FUNCTION_BLOCK "Qm"   // FB10, SCL
{ S7_Optimized_Access := 'FALSE' }
VERSION : 0.1
// Массовый расход
   VAR_INPUT
      Enable : Bool;   // Наличие параметра
      "a" : Real;   // Коэффициент расхода
      Ksh : Real;   // Поправочный коэффициент на шероховатость трубопровода
      Kp : Real;   // Поправочный коэффициент на неостроту входной кромки диафрагмы
      d : Real;   // Диаметр сужающего устройства при рабочих условиях (мм)
      ro : Real;   // Плотность среды в рабочих условиях (кг/м3)
      dP : Real;   // Перепад давления в рабочих условиях (кПа)
   END_VAR
   VAR_OUTPUT
      Value : Real;   // Значение массового расхода (т/ч)
   END_VAR
BEGIN
   (*Расход массового расхода (т/ч)*)
   IF #Enable THEN
       #Value := (#"a" * #Ksh * #Kp * 3.1415926 * SQR(#d / 1000) / 4) * SQRT(2 * #dP * 1000* #ro) * 3.6;
   ELSE
       #Value := 0;
   END_IF;
   IF #dP < 0 THEN
       #Value := 0;
   END_IF;
END_FUNCTION_BLOCK

FUNCTION_BLOCK "Qm_steam"   // FB11, SCL
{ S7_Optimized_Access := 'FALSE' }
VERSION : 0.1
// Массовый расход пара
   VAR_INPUT
      Enable : Bool;   // Наличие параметра
      "a" : Real;   // Коэффициент расхода
      Ksh : Real;   // Поправочный коэффициент на шероховатость трубопровода
      Kp : Real;   // Поправочный коэффициент на неостроту входной кромки диафрагмы
      d : Real;   // Диаметр сужающего устройства при рабочих условиях (мм)
      Dtrub : Real;   // Диаметр трубопровода при рабочих условиях (мм)
      k : Real;   // Показатель адиабаты
      ro : Real;   // Плотность среды в рабочих условиях (кг/м3)
      dP : Real;   // Перепад давления в рабочих условиях (кПа)
      P : Real;   // Давление в рабочих условиях (кПа)
   END_VAR
   VAR_OUTPUT
      Value : Real;   // Значение массового расхода (т/ч)
   END_VAR
   VAR
      "E" : Real;   // Коэффициент расширения
      B4 : Real;   // Относительный диаметр сужающего устройства (в 4 степени)
   END_VAR
BEGIN
   IF #Enable THEN
       (*Расчет относительного диаметра сужающего устройства (в 4 степени)*)
       #B4 := (#d /#Dtrub) ** 4;
       (*Расчет коэффициента расширения*)
       #"E" := 1 - ((0.351 + (0.256 * #B4) + (0.93 * SQR(#B4))) * (1 - ((1 - (#dP / #P)) ** (1 / #k))));
       #Value:= 0.25 * SQR(#d / 1000) * 3.1415926 * #"a" * #Ksh * #Kp * #"E" * SQRT(2 * #dP * #ro) * 3.6;
   ELSE
       #Value := 0;
   END_IF;
   IF #dP <= 0 OR #P <= 0 THEN
       #Value := 0;
   END_IF;
END_FUNCTION_BLOCK

FUNCTION_BLOCK "ro"   // FB12, SCL
{ S7_Optimized_Access := 'FALSE' }
VERSION : 0.1
// Расчет плотности
   VAR_INPUT
      P : Array[1..10] of Real;   // Давление (МПа)
      T : Array[1..20] of Real;   // Температура (град С)
      PT : Array[1..10, 1..20] of Real;   // Удельный объем (л/кг)
      Px : Real;   // Текущее давление (МПа)
      Tx : Real;   // Текущая температура (град С)
   END_VAR
   VAR_OUTPUT
      ro : Real;   // Значение удельной плотности (кг/м3)
   END_VAR
   VAR
      Pmin : Int;   // Нижняя граница текущего диапазона давления
      Pmax : Int;   // Верхняя граница текущего диапазона давления
      Tmin : Int;   // Нижняя граница текущего диапазона температуры
      Tmax : Int;   // Верхняя граница текущего диапазона температуры
      Pmin_Tmin : Real;   // Значение Pmin_Tmin рабочей области
      Pmin_Tmax : Real;   // Значение Pmin_Tmax рабочей области
      Pmax_Tmin : Real;   // Значение Pmax_Tmin рабочей области
      Pmax_Tmax : Real;   // Значение Pmax_Tmax рабочей области
      Px_Tmin : Real;   // Значение Px_Tmin суженной рабочей области
      Px_Tmax : Real;   // Значение Px_Tmax суженной рабочей области
      K_Px_Tmin : Real;
      B_Px_Tmin : Real;
      K_Px_Tmax : Real;
      B_Px_Tmax : Real;
      Px_Tx : Real;   // Искомое значение удельного объема (л/кг)
      K_Px_Tx : Real;
      B_Px_Tx : Real;
   END_VAR
BEGIN
   (*определение текущего диапазона давления*)
   IF #Px <= #P[2] THEN
       #Pmin := 1;
       #Pmax := 2;
   END_IF;
   IF #P[2] < #Px AND #Px <= #P[3] THEN
       #Pmin := 2;
       #Pmax := 3;
   END_IF;
   IF #P[3] < #Px AND #Px <= #P[4] THEN
       #Pmin := 3;
       #Pmax := 4;
   END_IF;
   IF #P[4] < #Px AND #Px <= #P[5] THEN
       #Pmin := 4;
       #Pmax := 5;
   END_IF;
   IF #P[5] < #Px AND #Px <= #P[6] THEN
       #Pmin := 5;
       #Pmax := 6;
   END_IF;
   IF #P[6] < #Px AND #Px <= #P[7] THEN
       #Pmin := 6;
       #Pmax := 7;
   END_IF;
   IF #P[7] < #Px AND #Px <= #P[8] THEN
       #Pmin := 7;
       #Pmax := 8;
   END_IF;
   IF #P[8] < #Px AND #Px <= #P[9] THEN
       #Pmin := 8;
       #Pmax := 9;
   END_IF;
   IF #P[9] < #Px THEN
       #Pmin := 9;
       #Pmax := 10;
   END_IF;

   (*определение текущего диапазона температуры*)
   IF #Tx <= #T[2] THEN
       #Tmin := 1;
       #Tmax := 2;
   END_IF;
   IF #T[2] < #Tx AND #Tx <= #T[3] THEN
       #Tmin := 2;
       #Tmax := 3;
   END_IF;
   IF #T[3] < #Tx AND #Tx <= #T[4] THEN
       #Tmin := 3;
       #Tmax := 4;
   END_IF;
   IF #T[4] < #Tx AND #Tx <= #T[5] THEN
       #Tmin := 4;
       #Tmax := 5;
   END_IF;
   IF #T[5] < #Tx AND #Tx <= #T[6] THEN
       #Tmin := 5;
       #Tmax := 6;
   END_IF;
   IF #T[6] < #Tx AND #Tx <= #T[7] THEN
       #Tmin := 6;
       #Tmax := 7;
   END_IF;
   IF #T[7] < #Tx AND #Tx <= #T[8] THEN
       #Tmin := 7;
       #Tmax := 8;
   END_IF;
   IF #T[8] < #Tx AND #Tx <= #T[9] THEN
       #Tmin := 8;
       #Tmax := 9;
   END_IF;
   IF #T[9] < #Tx AND #Tx <= #T[10] THEN
       #Tmin := 9;
       #Tmax := 10;
   END_IF;
   IF #T[10] < #Tx AND #Tx <= #T[11] THEN
       #Tmin := 10;
       #Tmax := 11;
   END_IF;
   IF #T[11] < #Tx AND #Tx <= #T[12] THEN
       #Tmin := 11;
       #Tmax := 12;
   END_IF;
   IF #T[12] < #Tx AND #Tx <= #T[13] THEN
       #Tmin := 12;
       #Tmax := 13;
   END_IF;
   IF #T[13] < #Tx AND #Tx <= #T[14] THEN
       #Tmin := 13;
       #Tmax := 14;
   END_IF;
   IF #T[14] < #Tx AND #Tx <= #T[15] THEN
       #Tmin := 14;
       #Tmax := 15;
   END_IF;
   IF #T[15] < #Tx AND #Tx <= #T[16] THEN
       #Tmin := 15;
       #Tmax := 16;
   END_IF;
   IF #T[16] < #Tx AND #Tx <= #T[17] THEN
       #Tmin := 16;
       #Tmax := 17;
   END_IF;
   IF #T[17] < #Tx AND #Tx <= #T[18] THEN
       #Tmin := 17;
       #Tmax := 18;
   END_IF;
   IF #T[18] < #Tx AND #Tx <= #T[19] THEN
       #Tmin := 18;
       #Tmax := 19;
   END_IF;
   IF #T[19] < #Tx THEN
       #Tmin := 19;
       #Tmax := 20;
   END_IF;

   (*определение рабочей области*)
   #Pmin_Tmin := #PT[#Pmin, #Tmin];
   #Pmin_Tmax := #PT[#Pmin, #Tmax];
   #Pmax_Tmin := #PT[#Pmax, #Tmin];
   #Pmax_Tmax := #PT[#Pmax, #Tmax];

   (*определение суженной по давлению рабочей области*)
   #K_Px_Tmin := (#Pmax_Tmin - #Pmin_Tmin) / (#P[#Pmax] - #P[#Pmin]);
   #B_Px_Tmin := #Pmin_Tmin - #K_Px_Tmin * #P[#Pmin];
   #Px_Tmin := #K_Px_Tmin * #Px + #B_Px_Tmin;

   #K_Px_Tmax := (#Pmax_Tmax - #Pmin_Tmax) / (#P[#Pmax] - #P[#Pmin]);
   #B_Px_Tmax := #Pmin_Tmax - #K_Px_Tmax * #P[#Pmin];
   #Px_Tmax := #K_Px_Tmax * #Px + #B_Px_Tmax;

   (*определение искомого значения удельного объема*)
   #K_Px_Tx := (#Px_Tmax - #Px_Tmin) / (#T[#Tmax] - #T[#Tmin]);
   #B_Px_Tx := #Px_Tmin - #K_Px_Tx * #T[#Tmin];
   #Px_Tx := #K_Px_Tx * #Tx + #B_Px_Tx;

   (*определение значения удельной плотности*)
   #ro := 1000 / #Px_Tx;
END_FUNCTION_BLOCK

FUNCTION_BLOCK "Qs"   // FB13, SCL
{ S7_Optimized_Access := 'FALSE' }
VERSION : 0.1
// Расход приведенный к стандартным условиям (нм3/ч)
   VAR_INPUT
      P : Real;   // Давление в рабочих условиях (Па)
      Q : Real;   // Объемный расход измеренный (м3/ч)
      T : Real;   // Температура в рабочих условиях (град С)
      ro_c : Real;   // Плотность при стандартных условиях (кг/м3)
      Xa : Real;   // молярная/объемная доля азота (в долях от 1)
      Xy : Real;   // молярная/объемная доля диоксида углерода (в долях от 1)
   END_VAR
   VAR_OUTPUT
      Qs : Real;   // Объемный расход приведенный к стандартным условиям (нм3/ч)
   END_VAR
   VAR
      K : Real;   // коэффициент сжимаемости
      Z : Real;   // фактор сжимаемости при рабочих условиях
      Zc : Real;   // фактор сжимаемости при стандартных условиях
      Tpk : Real;
      Ppk : Real;
      Ta : Real;
      Pa : Real;
      dTa : Real;
      F : Real;   // Корректирующий множитель
      Theta1 : Real;
      Theta0 : Real;
      B0 : Real;
      B1 : Real;
      B2 : Real;
   END_VAR
BEGIN
   (*расчет фактора сжимаемости при стандартных условиях*)
   #Zc := 1 - SQR(0.0741*#ro_c-0.006-0.063*#Xa-0.0575*#Xy);

   (*расчет фактора сжимаемости при рабочих условиях*)
   #Tpk:=88.25*(0.9915+1.759*#ro_c-#Xy-1.681*#Xa);
   #Ppk := 2.9585 * (1.608-0.05994*#ro_c+#Xy-0.392*#Xa);

   #Ta := 0.71892 * ((#T + 273.15)/ #Tpk) + 0.0007;
   #Pa := 0.6714 * (#P / (1000000*#Ppk)) + 0.0147;

   #dTa := #Ta - 1.09;

   //расчет корректирующего множителя
   IF 0 <= #Pa AND #Pa <= 2 AND 0 <= #dTa AND #dTa <= 0.3 THEN
       #F := (0.00075 * (#Pa ** 2.3)) / (2.718281828459045 ** (20 * #dTa)) + 0.0011*SQRT(#dTa)*SQR((#Pa*(2.17-#Pa+1.4*SQRT(#dTa))));
   END_IF;
   IF 0 <= #Pa AND #Pa < 1.3 AND -0.25 <= #dTa AND #dTa < 0 THEN
       #F := 0.00075 * (#Pa ** 2.3) * (2 - (2.718281828459045 ** (20 * #dTa))) + 1.317 * #Pa * (1.69 - SQR(#Pa)) * (#dTa ** 4);
   END_IF;
   IF 1.3 <= #Pa AND #Pa < 2 AND -0.21 <= #dTa AND #dTa < 0 THEN
       #F := 0.00075 * (#Pa ** 2.3) * (2 - (2.718281828459045 ** (20 * #dTa)))+0.455*#Pa*(1.3-#Pa)*(4.0195200-SQR(#Pa))*(#dTa*(0.03249+18.028*SQR(#dTa))+SQR(#dTa)*(2.0167+SQR(#dTa)*(42.844+200*SQR(#dTa))));
   END_IF;

   #Theta1 := (#Ta ** 5) / (SQR(#Ta)*(6.60756*#Ta-4.42646)+3.22706);
   #Theta0 := ((SQR(#Ta)*(1.77218-0.8879*#Ta)+0.305131) * #Theta1) / (#Ta ** 4);
   #B1 := ((2 * #Theta1) / 3) - SQR(#Theta0);
   #B0 := #Theta0 * (#Theta1 - SQR(#Theta0)) + 0.1 * #Theta1 * #Pa * (#F - 1);
   #B2 := (#B0 + SQRT(SQR(#B0) + #B1 ** 3)) ** (0.333334);

   #Z := ((1+(0.00132/(#Ta**3.25))) / ((#B1/#B2)-#B2+#Theta0)) * (#Pa / 10);

   (*расчет коэффициента сжимаемости*)
   #K := #Z / #Zc;

   (*расчет объемного расхода приведенного к стандартным условиям (нм3/ч)*)
   #Qs := ((#P+101325) * 293.15 * #Q) / (101325 * (#T + 273.15) * #K);
END_FUNCTION_BLOCK

FUNCTION "Read_inputs" : Void   // FC1, SCL
{ S7_Optimized_Access := 'TRUE' }
VERSION : 0.1
BEGIN
   (*ЧТЕНИЕ ВХОДОВ*)
   (*Чтение аналоговых входов*)
   //Температура питательной воды перед экономайзером
   "T_water_before_economizer"();
   //Температура питательной воды после экономайзера
   "T_water_after_economizer"();
   //Перепад давления питательной воды на котел
   "dP_water_boiler"();
   //Давление питательной воды до регулятора
   "P_water_before_regul"();
   //Давление питательной воды после регулятора
   "P_water_after_regul"();
   //Перепад давления пара в магистраль
   "dP_steam"();
   //Давление пара в барабане
   "P_steam"();
   //Разрежение в топке котла
   "dP_furnace_boiler"();
   //Давление газа между ПЗК-1 и ПЗК-2
   "P_gas_between_PZK1_and_PZK2"();
   //Давление газа перед горелкой
   "P_gas_before_burner"();
   //Давление воздуха к горелке
   "P_air_burner"();
   //Положение рег. заслонки питательной воды на котел
   "ZRW_position"();
   //Положение рег. заслонки газа перед котлом
   "ZRG_position"();
   //Положение направл. аппарата вентилятора
   "NAV_position"();
   //Положение направл. аппарата дымососа
   "NAD_position"();
   //Температура уходящих дымовых газов  перед экономайзером
   "T_exhaust_gas_before_economizer"();
   //Температура уходящих дымовых газов  после экономайзера
   "T_exhaust_gas_after_economizer"();
   //Разрежение в дымоходе перед экономайзером
   "dP_exhaust_gas_before_economizer"();
   //Разрежение в дымоходе после экономайзера
   "dP_exhaust_gas_after_economizer"();
   //Давление газа перед БГ
   "P_gas_before_BG"();
   //Температура газа перед БГ
   "T_gas_before_BG"();
   //Давление пара в магистраль
   "P_steam_pipe"();
   //Температура пара в магистраль
   "T_steam"();
   //Текущее значение частоты ПЧ вентилятора
   "DV_current_frequency"();
   //Текущее значение частоты ПЧ дымососа
   "DS_current_frequency"();
   //Перепад давления на измерительной колонке 
   "dP_water_level"();
   //Уровень воды в измерительной колонке
   "L_water_level"(LL_ADC_new := "dP_water_level".LL_ADC_new,
                   HL_ADC_new := "dP_water_level".HL_ADC_new,
                   Apply_new_limit := "dP_water_level".Apply_new_limit);
   //Уровень воды в барабане
   "L_water"(LL_sensor_new := "L_water_level".LL_sensor_new + "Technology".Offset_level_water,
             HL_sensor_new := "L_water_level".HL_sensor_new + "Technology".Offset_level_water,
             LL_ADC_new := "dP_water_level".LL_ADC_new,
             HL_ADC_new := "dP_water_level".HL_ADC_new,
             Apply_new_limit := "dP_water_level".Apply_new_limit);

   (*Чтение дискретных входов*)
   //Наличие пламени горелки
   "Burner_flame"();
   //Наличие пламени запальника горелки
   "Igniter_flame"();
   //Клапан безопасности закрыт
   "KB_close"();
   //Клапан опрессовки открыт
   "KO_open"();
   //Клапан запальника открыт
   "KZ_open"();
   //ПЗК-1 горелки открыт
   "PZK1_open"();
   //ПЗК-2 горелки не закрыт
   "PZK2_not_close"();
   //Давление газа перед БГ мин.
   "P_gas_before_BG_min"();
   //Давление газа перед БГ макс.
   "P_gas_before_BG_max"();
   //Давление воздуха перед горелкой мин.
   "P_air_before_burner_min"();
   //Давление газа перед горелкой мин.
   "P_gas_before_burner_min"();
   //Давление газа перед горелкой макс.
   "P_gas_before_burner_max"();
   //Регулирующая заслонка газа открыта
   "ZRG_open"();
   //Регулирующая заслонка газа закрыта
   "ZRG_close"();
   //Регулирующая заслонка газа среднее
   "ZRG_middle"();
   //Регулирующая заслонка газа. БРУ в положении "Авт"
   "ZRG_avto"();
   //НАВ открыт
   "NAV_open"();
   //НАВ закрыт
   "NAV_close"();
   //НАВ среднее
   "NAV_middle"();
   //НАВ. БРУ в положении "Авт"
   "NAV_avto"();
   //НАД открыт
   "NAD_open"();
   //НАД закрыт
   "NAD_close"();
   //НАД среднее
   "NAD_middle"();
   //НАД. БРУ в положении "Авт"
   "NAD_avto"();
   //ПЗК-2 горелки открыт
   "PZK2_open"();
   //Разрежение в топке котла мин.
   "dP_furnace_boiler_min"();
   //Давление питательной воды после регулятора мин.
   "P_water_after_regul_min"();
   //Давление пара в барабане макс.
   "P_steam_max"();
   //Уровень воды в барабане мин.
   "L_water_min"();
   //Уровень воды в барабане макс.
   "L_water_max"();
   //Вызов к шкафу электропитания
   "Call_power_supply_cabinet"();
   //Авария ПЧ ДВ
   "DV_Invertor_alarm"();
   //Режим работы ДВ «Местный»
   "DV_local_control"();
   //Режим работы ДВ «Дистанционный»
   "DV_dist_control"();
   //Режим "СЕТЬ" ДВ
   "DV_powergrid_mode"();
   //Режим "ПЧ" ДВ
   "DV_invertor_mode"();
   //Автомат работы ДВ от ПЧ включен
   "DV_invertor_QF_on"();
   //Автомат работы ДВ от сети включен
   "DV_powergrid_QF_on"();
   //Включен ДВ от ПЧ
   "DV_invertor_on"();
   //Включен ДВ от сети
   "DV_powergrid_on"();
   //Нет напряжения сети ШУД ДВ
   "DV_no_voltage"();
   //Авария ПЧ ДС
   "DS_Invertor_alarm"();
   //Режим работы ДС «Местный»
   "DS_local_control"();
   //Режим работы ДC «Дистанционный»
   "DS_dist_control"();
   //Режим "СЕТЬ" ДC
   "DS_powergrid_mode"();
   //Режим "ПЧ" ДС
   "DS_invertor_mode"();
   //Автомат работы ДС от ПЧ включен
   "DS_invertor_QF_on"();
   //Автомат работы ДС от сети включен
   "DS_powergrid_QF_on"();
   //Включен ДС от ПЧ
   "DS_invertor_on"();
   //Включен ДС от сети
   "DS_powergrid_on"();
   //Нет напряжения сети ШУД ДС
   "DS_no_voltage"();
   //Загазованность СО I порог
   "CO_1"();
   //Загазованность СО II порог
   "CO_2"();
   //Загазованность CH4 порог
   "CH4"();
   //Кнопка СТОП
   "Btn_STOP"();
   //Кнопка Вентиляция
   "Btn_Ventilation"();
   //Кнопка Розжиг
   "Btn_Ignition"();
   //Кнопка Сброс звука / Проверка звука
   "Btn_Sound"();
   //Регулирующая заслонка питательной воды на котел открыта
   "ZRW_open"();
   //Регулирующая заслонка питательной воды на котел закрыта
   "ZRW_close"();
   //Регулирующая заслонка питательной воды на котел среднее
   "ZRW_middle"();
   //Регулирующая заслонка питательной воды на котел. БРУ в положении "Авт"
   "ZRW_avto"();
   //Питание контроллера от ИБП
   "Power_PLC_from_UPS"();
   //Заряд батареи ИБП низкий
   "UPS_Low_charge"();
   //ЗРГ Напряжение в норме
   "ZRG_voltage_ok"();
   //НАВ Напряжение в норме
   "NAV_voltage_ok"();
   //НАД Напряжение в норме
   "NAD_voltage_ok"();
   //ЗРВ Напряжение в норме
   "ZRW_voltage_ok"();
   //Контроль питания сети ~400В 1ШЭУ
   "SHEU_voltage_ok"();
   //ЗДГ перед БГ. не открыта
   "ZDG_no_open"();
   //ЗДГ перед БГ. не закрыта
   "ZDG_no_close"();
   //ЗДГ перед БГ. ход открытие
   "ZDG_opening"();
   //ЗДГ перед БГ. ход закрытие
   "ZDG_closing"();
   //ЗДГ перед БГ. Напряжение в норме
   "ZDG_voltage_ok"();
   //ЗДСВ перед котлом. не открыта
   "ZDSV_before_boiler_no_open"();
   //ЗДСВ перед котлом. не закрыта
   "ZDSV_before_boiler_no_close"();
   //ЗДСВ перед котлом. ход открытие
   "ZDSV_before_boiler_opening"();
   //ЗДСВ перед котлом. ход закрытие
   "ZDSV_before_boiler_closing"();
   //ЗДСВ перед котлом. Напряжение в норме
   "ZDSV_before_boiler_voltage_ok"();
   //ЗДСВ перед котлом. ограничитель крутящего момента
   "ZDSV_before_boiler_limit_rotational_moment"();
   //ГПЗ. не открыта
   "GPZ_no_open"();
   //ГПЗ. не закрыта
   "GPZ_no_close"();
   //ГПЗ. ход открытие
   "GPZ_opening"();
   //ГПЗ. ход закрытие
   "GPZ_closing"();
   //ГПЗ. Напряжение в норме
   "GPZ_voltage_ok"();
   //ГПЗ. ограничитель крутящего момента
   "GPZ_limit_rotational_moment"();

   (*Контроль питания ~400В резервной горелки, статус «Работа на дизтопливе»

   Режим работы резервной горелки

   Блокировка пламени резервной горелки

   Режим “Большое пламя» резервной горелки*)

   //Расход газа (м3/ч)
   //"Q_gas".scale_unit := (293.15 * INT_TO_REAL("Technology".Q_gas_scale_unit) * ("P_gas_before_BG".Value/1000.0 + "Technology".P_atm))/(0.101325*(273.15 + "T_gas_before_BG".Value)*"Technology".K_gas);
   "Q_gas"();

   //Расход газа приведенного к стандартным условиям (нм3/ч)
   "Qs_gas"(P := "P_gas_before_BG".Value * 1000,
            Q := "Q_gas".moment_consumption,
            T := "T_gas_before_BG".Value);

   //Массовый расход воды
   "Q_water"(dP := "dP_water_boiler".Value);

   //плотность пара
   "ro_steam"(Px := ("P_steam_pipe".Value) / 10,
              Tx := "T_steam".Value);

   //Массовый расход пара
   IF "GPZ_no_close".Value THEN
       "Q_steam"(dP := "dP_steam".Value * 1000,
                 P := ("P_steam_pipe".Value + 1) * 100000,
                 ro := "ro_steam".ro);
   ELSE
       "Q_steam"(dP := 0 * 1000,
                 P := ("P_steam_pipe".Value + 1) * 100000,
                 ro := "ro_steam".ro);
   END_IF;
   "Q1_water".Value := ("Qs_gas".Qs * "Q1_water".Calorie * "Q1_water".KPD) / ("Q1_water"."E" * 1000);

   (*настройка датчиков уровня*)
   "dP_main" := ((("dP_water_boiler".HL_sensor - "dP_water_boiler".LL_sensor) / INT_TO_REAL(27648 - 0)) * INT_TO_REAL("Module03Chanel5_AI")) + "dP_water_boiler".LL_sensor;
   "L_main" := ((("L_water".HL_sensor - "L_water".LL_sensor) / INT_TO_REAL(0 - 27648)) * INT_TO_REAL("Module03Chanel5_AI")) + "L_water".HL_sensor;
   "Current_main" := (((20 - 4) / (INT_TO_REAL(27648 - 0))) * (INT_TO_REAL("Module03Chanel5_AI"))) + 4;

   "dP_res" := ((("dP_water_boiler".HL_sensor - "dP_water_boiler".LL_sensor) / INT_TO_REAL(27648 - 0)) * INT_TO_REAL("Module04Chanel5_AI")) + "dP_water_boiler".LL_sensor;
   "L_res" := ((("L_water".HL_sensor - "L_water".LL_sensor) / INT_TO_REAL(0 - 27648)) * INT_TO_REAL("Module04Chanel5_AI")) + "L_water".HL_sensor;
   "Current_res" := (((20 - 4) / (INT_TO_REAL(27648 - 0))) * (INT_TO_REAL("Module04Chanel5_AI"))) + 4;

   //подмена дискретных входов
   "Module12Chanel1_DI" := "Module12Chanel1_DO";
   "Module12Chanel2_DI" := "Module12Chanel2_DO";
   "Module12Chanel3_DI" := "Module12Chanel3_DO";
   "Module12Chanel4_DI" := "Module12Chanel4_DO";
   "Module12Chanel5_DI" := "Module12Chanel5_DO";
   "Module12Chanel6_DI" := "Module12Chanel6_DO";
   "Module12Chanel7_DI" := "Module12Chanel7_DO";
   "Module12Chanel8_DI" := "Module12Chanel8_DO";
   "Module12Chanel9_DI" := "Module12Chanel9_DO";
   "Module12Chanel10_DI" := "Module12Chanel10_DO";
   "Module12Chanel11_DI" := "Module12Chanel11_DO";
   "Module12Chanel12_DI" := "Module12Chanel12_DO";
   "Module12Chanel13_DI" := "Module12Chanel13_DO";
   "Module12Chanel14_DI" := "Module12Chanel14_DO";
   "Module12Chanel15_DI" := "Module12Chanel15_DO";
   "Module12Chanel16_DI" := "Module12Chanel16_DO";
END_FUNCTION

FUNCTION "read_discret" : Bool   // FC2, SCL
{ S7_Optimized_Access := 'TRUE' }
AUTHOR : Dmitriy_Petrov
VERSION : 0.1
// Функция чтения дискретного параметра
   VAR_INPUT
      Invert : Bool;   // Инвертирование сигнала
   END_VAR
   VAR_IN_OUT
      N_module : USInt;   // № модуля (начиная с 1)
      N_chanel : USInt;   // № канала (начиная с 1)
   END_VAR
   VAR_TEMP
      Signal : Bool;   // Значение сигнала
   END_VAR
   // Ret_Val : Текущее значение
BEGIN
   (*проверка правильности введеного значения № Модуля*)
   IF #N_module < 1 OR #N_module > 25 THEN
       #N_module := 0;
   END_IF;

   (*проверка правильности введеного значения № Канала*)
   IF #N_module = 0 THEN
       #N_chanel := 0;
   ELSE
       IF #N_chanel < 1 OR #N_chanel > 16 THEN
           #N_chanel := 0;
       END_IF;
   END_IF;

   (*считывание и обработка дискретного сигнала с выбранного канала*)
   CASE #N_module OF
       1:  // Модуль 1
           CASE #N_chanel OF
               1:
                   #Signal := "Module01Chanel1_DI";   //Канал 1
               2:
                   #Signal := "Module01Chanel2_DI";   //Канал 2
               3:
                   #Signal := "Module01Chanel3_DI";   //Канал 3
               4:
                   #Signal := "Module01Chanel4_DI";   //Канал 4
               5:
                   #Signal := "Module01Chanel5_DI";   //Канал 5
               6:
                   #Signal := "Module01Chanel6_DI";   //Канал 6
               7:
                   #Signal := "Module01Chanel7_DI";   //Канал 7
               8:
                   #Signal := "Module01Chanel8_DI";   //Канал 8
               9:
                   #Signal := "Module01Chanel9_DI";   //Канал 9
               10:
                   #Signal := "Module01Chanel10_DI";  //Канал 10
               11:
                   #Signal := "Module01Chanel11_DI";  //Канал 11
               12:
                   #Signal := "Module01Chanel12_DI";  //Канал 12
               13:
                   #Signal := "Module01Chanel13_DI";  //Канал 13
               14:
                   #Signal := "Module01Chanel14_DI";  //Канал 14
               15:
                   #Signal := "Module01Chanel15_DI";  //Канал 15
               16:
                   #Signal := "Module01Chanel16_DI";  //Канал 16
               ELSE
                   #Signal := FALSE;
           END_CASE;
       2:  // Модуль 2
           CASE #N_chanel OF
               1:
                   #Signal := "Module02Chanel1_DI";   //Канал 1
               2:
                   #Signal := "Module02Chanel2_DI";   //Канал 2
               3:
                   #Signal := "Module02Chanel3_DI";   //Канал 3
               4:
                   #Signal := "Module02Chanel4_DI";   //Канал 4
               5:
                   #Signal := "Module02Chanel5_DI";   //Канал 5
               6:
                   #Signal := "Module02Chanel6_DI";   //Канал 6
               7:
                   #Signal := "Module02Chanel7_DI";   //Канал 7
               8:
                   #Signal := "Module02Chanel8_DI";   //Канал 8
               9:
                   #Signal := "Module02Chanel9_DI";   //Канал 9
               10:
                   #Signal := "Module02Chanel10_DI";  //Канал 10
               11:
                   #Signal := "Module02Chanel11_DI";  //Канал 11
               12:
                   #Signal := "Module02Chanel12_DI";  //Канал 12
               13:
                   #Signal := "Module02Chanel13_DI";  //Канал 13
               14:
                   #Signal := "Module02Chanel14_DI";  //Канал 14
               15:
                   #Signal := "Module02Chanel15_DI";  //Канал 15
               16:
                   #Signal := "Module02Chanel16_DI";  //Канал 16
               ELSE
                   #Signal := FALSE;
           END_CASE;
       3:  // Модуль 3
           CASE #N_chanel OF
               1:
                   #Signal := "Module03Chanel1_DI";   //Канал 1
               2:
                   #Signal := "Module03Chanel2_DI";   //Канал 2
               3:
                   #Signal := "Module03Chanel3_DI";   //Канал 3
               4:
                   #Signal := "Module03Chanel4_DI";   //Канал 4
               5:
                   #Signal := "Module03Chanel5_DI";   //Канал 5
               6:
                   #Signal := "Module03Chanel6_DI";   //Канал 6
               7:
                   #Signal := "Module03Chanel7_DI";   //Канал 7
               8:
                   #Signal := "Module03Chanel8_DI";   //Канал 8
               9:
                   #Signal := "Module03Chanel9_DI";   //Канал 9
               10:
                   #Signal := "Module03Chanel10_DI";  //Канал 10
               11:
                   #Signal := "Module03Chanel11_DI";  //Канал 11
               12:
                   #Signal := "Module03Chanel12_DI";  //Канал 12
               13:
                   #Signal := "Module03Chanel13_DI";  //Канал 13
               14:
                   #Signal := "Module03Chanel14_DI";  //Канал 14
               15:
                   #Signal := "Module03Chanel15_DI";  //Канал 15
               16:
                   #Signal := "Module03Chanel16_DI";  //Канал 16
               ELSE
                   #Signal := FALSE;
           END_CASE;
       4:  // Модуль 4
           CASE #N_chanel OF
               1:
                   #Signal := "Module04Chanel1_DI";   //Канал 1
               2:
                   #Signal := "Module04Chanel2_DI";   //Канал 2
               3:
                   #Signal := "Module04Chanel3_DI";   //Канал 3
               4:
                   #Signal := "Module04Chanel4_DI";   //Канал 4
               5:
                   #Signal := "Module04Chanel5_DI";   //Канал 5
               6:
                   #Signal := "Module04Chanel6_DI";   //Канал 6
               7:
                   #Signal := "Module04Chanel7_DI";   //Канал 7
               8:
                   #Signal := "Module04Chanel8_DI";   //Канал 8
               9:
                   #Signal := "Module04Chanel9_DI";   //Канал 9
               10:
                   #Signal := "Module04Chanel10_DI";  //Канал 10
               11:
                   #Signal := "Module04Chanel11_DI";  //Канал 11
               12:
                   #Signal := "Module04Chanel12_DI";  //Канал 12
               13:
                   #Signal := "Module04Chanel13_DI";  //Канал 13
               14:
                   #Signal := "Module04Chanel14_DI";  //Канал 14
               15:
                   #Signal := "Module04Chanel15_DI";  //Канал 15
               16:
                   #Signal := "Module04Chanel16_DI";  //Канал 16
               ELSE
                   #Signal := FALSE;
           END_CASE;
       5:  // Модуль 5
           CASE #N_chanel OF
               1:
                   #Signal := "Module05Chanel1_DI";   //Канал 1
               2:
                   #Signal := "Module05Chanel2_DI";   //Канал 2
               3:
                   #Signal := "Module05Chanel3_DI";   //Канал 3
               4:
                   #Signal := "Module05Chanel4_DI";   //Канал 4
               5:
                   #Signal := "Module05Chanel5_DI";   //Канал 5
               6:
                   #Signal := "Module05Chanel6_DI";   //Канал 6
               7:
                   #Signal := "Module05Chanel7_DI";   //Канал 7
               8:
                   #Signal := "Module05Chanel8_DI";   //Канал 8
               9:
                   #Signal := "Module05Chanel9_DI";   //Канал 9
               10:
                   #Signal := "Module05Chanel10_DI";  //Канал 10
               11:
                   #Signal := "Module05Chanel11_DI";  //Канал 11
               12:
                   #Signal := "Module05Chanel12_DI";  //Канал 12
               13:
                   #Signal := "Module05Chanel13_DI";  //Канал 13
               14:
                   #Signal := "Module05Chanel14_DI";  //Канал 14
               15:
                   #Signal := "Module05Chanel15_DI";  //Канал 15
               16:
                   #Signal := "Module05Chanel16_DI";  //Канал 16
               ELSE
                   #Signal := FALSE;
           END_CASE;
       6:  // Модуль 6
           CASE #N_chanel OF
               1:
                   #Signal := "Module06Chanel1_DI";   //Канал 1
               2:
                   #Signal := "Module06Chanel2_DI";   //Канал 2
               3:
                   #Signal := "Module06Chanel3_DI";   //Канал 3
               4:
                   #Signal := "Module06Chanel4_DI";   //Канал 4
               5:
                   #Signal := "Module06Chanel5_DI";   //Канал 5
               6:
                   #Signal := "Module06Chanel6_DI";   //Канал 6
               7:
                   #Signal := "Module06Chanel7_DI";   //Канал 7
               8:
                   #Signal := "Module06Chanel8_DI";   //Канал 8
               9:
                   #Signal := "Module06Chanel9_DI";   //Канал 9
               10:
                   #Signal := "Module06Chanel10_DI";  //Канал 10
               11:
                   #Signal := "Module06Chanel11_DI";  //Канал 11
               12:
                   #Signal := "Module06Chanel12_DI";  //Канал 12
               13:
                   #Signal := "Module06Chanel13_DI";  //Канал 13
               14:
                   #Signal := "Module06Chanel14_DI";  //Канал 14
               15:
                   #Signal := "Module06Chanel15_DI";  //Канал 15
               16:
                   #Signal := "Module06Chanel16_DI";  //Канал 16
               ELSE
                   #Signal := FALSE;
           END_CASE;
       7:  // Модуль 7
           CASE #N_chanel OF
               1:
                   #Signal := "Module07Chanel1_DI";   //Канал 1
               2:
                   #Signal := "Module07Chanel2_DI";   //Канал 2
               3:
                   #Signal := "Module07Chanel3_DI";   //Канал 3
               4:
                   #Signal := "Module07Chanel4_DI";   //Канал 4
               5:
                   #Signal := "Module07Chanel5_DI";   //Канал 5
               6:
                   #Signal := "Module07Chanel6_DI";   //Канал 6
               7:
                   #Signal := "Module07Chanel7_DI";   //Канал 7
               8:
                   #Signal := "Module07Chanel8_DI";   //Канал 8
               9:
                   #Signal := "Module07Chanel9_DI";   //Канал 9
               10:
                   #Signal := "Module07Chanel10_DI";  //Канал 10
               11:
                   #Signal := "Module07Chanel11_DI";  //Канал 11
               12:
                   #Signal := "Module07Chanel12_DI";  //Канал 12
               13:
                   #Signal := "Module07Chanel13_DI";  //Канал 13
               14:
                   #Signal := "Module07Chanel14_DI";  //Канал 14
               15:
                   #Signal := "Module07Chanel15_DI";  //Канал 15
               16:
                   #Signal := "Module07Chanel16_DI";  //Канал 16
               ELSE
                   #Signal := FALSE;
           END_CASE;
       8:  // Модуль 8
           CASE #N_chanel OF
               1:
                   #Signal := "Module08Chanel1_DI";   //Канал 1
               2:
                   #Signal := "Module08Chanel2_DI";   //Канал 2
               3:
                   #Signal := "Module08Chanel3_DI";   //Канал 3
               4:
                   #Signal := "Module08Chanel4_DI";   //Канал 4
               5:
                   #Signal := "Module08Chanel5_DI";   //Канал 5
               6:
                   #Signal := "Module08Chanel6_DI";   //Канал 6
               7:
                   #Signal := "Module08Chanel7_DI";   //Канал 7
               8:
                   #Signal := "Module08Chanel8_DI";   //Канал 8
               9:
                   #Signal := "Module08Chanel9_DI";   //Канал 9
               10:
                   #Signal := "Module08Chanel10_DI";  //Канал 10
               11:
                   #Signal := "Module08Chanel11_DI";  //Канал 11
               12:
                   #Signal := "Module08Chanel12_DI";  //Канал 12
               13:
                   #Signal := "Module08Chanel13_DI";  //Канал 13
               14:
                   #Signal := "Module08Chanel14_DI";  //Канал 14
               15:
                   #Signal := "Module08Chanel15_DI";  //Канал 15
               16:
                   #Signal := "Module08Chanel16_DI";  //Канал 16
               ELSE
                   #Signal := FALSE;
           END_CASE;
       9:  // Модуль 9
           CASE #N_chanel OF
               1:
                   #Signal := "Module09Chanel1_DI";   //Канал 1
               2:
                   #Signal := "Module09Chanel2_DI";   //Канал 2
               3:
                   #Signal := "Module09Chanel3_DI";   //Канал 3
               4:
                   #Signal := "Module09Chanel4_DI";   //Канал 4
               5:
                   #Signal := "Module09Chanel5_DI";   //Канал 5
               6:
                   #Signal := "Module09Chanel6_DI";   //Канал 6
               7:
                   #Signal := "Module09Chanel7_DI";   //Канал 7
               8:
                   #Signal := "Module09Chanel8_DI";   //Канал 8
               9:
                   #Signal := "Module09Chanel9_DI";   //Канал 9
               10:
                   #Signal := "Module09Chanel10_DI";  //Канал 10
               11:
                   #Signal := "Module09Chanel11_DI";  //Канал 11
               12:
                   #Signal := "Module09Chanel12_DI";  //Канал 12
               13:
                   #Signal := "Module09Chanel13_DI";  //Канал 13
               14:
                   #Signal := "Module09Chanel14_DI";  //Канал 14
               15:
                   #Signal := "Module09Chanel15_DI";  //Канал 15
               16:
                   #Signal := "Module09Chanel16_DI";  //Канал 16
               ELSE
                   #Signal := FALSE;
           END_CASE;
       10:  // Модуль 10
           CASE #N_chanel OF
               1:
                   #Signal := "Module10Chanel1_DI";   //Канал 1
               2:
                   #Signal := "Module10Chanel2_DI";   //Канал 2
               3:
                   #Signal := "Module10Chanel3_DI";   //Канал 3
               4:
                   #Signal := "Module10Chanel4_DI";   //Канал 4
               5:
                   #Signal := "Module10Chanel5_DI";   //Канал 5
               6:
                   #Signal := "Module10Chanel6_DI";   //Канал 6
               7:
                   #Signal := "Module10Chanel7_DI";   //Канал 7
               8:
                   #Signal := "Module10Chanel8_DI";   //Канал 8
               9:
                   #Signal := "Module10Chanel9_DI";   //Канал 9
               10:
                   #Signal := "Module10Chanel10_DI";  //Канал 10
               11:
                   #Signal := "Module10Chanel11_DI";  //Канал 11
               12:
                   #Signal := "Module10Chanel12_DI";  //Канал 12
               13:
                   #Signal := "Module10Chanel13_DI";  //Канал 13
               14:
                   #Signal := "Module10Chanel14_DI";  //Канал 14
               15:
                   #Signal := "Module10Chanel15_DI";  //Канал 15
               16:
                   #Signal := "Module10Chanel16_DI";  //Канал 16
               ELSE
                   #Signal := FALSE;
           END_CASE;
       11:  // Модуль 11
           CASE #N_chanel OF
               1:
                   #Signal := "Module11Chanel1_DI";   //Канал 1
               2:
                   #Signal := "Module11Chanel2_DI";   //Канал 2
               3:
                   #Signal := "Module11Chanel3_DI";   //Канал 3
               4:
                   #Signal := "Module11Chanel4_DI";   //Канал 4
               5:
                   #Signal := "Module11Chanel5_DI";   //Канал 5
               6:
                   #Signal := "Module11Chanel6_DI";   //Канал 6
               7:
                   #Signal := "Module11Chanel7_DI";   //Канал 7
               8:
                   #Signal := "Module11Chanel8_DI";   //Канал 8
               9:
                   #Signal := "Module11Chanel9_DI";   //Канал 9
               10:
                   #Signal := "Module11Chanel10_DI";  //Канал 10
               11:
                   #Signal := "Module11Chanel11_DI";  //Канал 11
               12:
                   #Signal := "Module11Chanel12_DI";  //Канал 12
               13:
                   #Signal := "Module11Chanel13_DI";  //Канал 13
               14:
                   #Signal := "Module11Chanel14_DI";  //Канал 14
               15:
                   #Signal := "Module11Chanel15_DI";  //Канал 15
               16:
                   #Signal := "Module11Chanel16_DI";  //Канал 16
               ELSE
                   #Signal := FALSE;
           END_CASE;
       12:  // Модуль 12
           CASE #N_chanel OF
               1:
                   #Signal := "Module12Chanel1_DI";   //Канал 1
               2:
                   #Signal := "Module12Chanel2_DI";   //Канал 2
               3:
                   #Signal := "Module12Chanel3_DI";   //Канал 3
               4:
                   #Signal := "Module12Chanel4_DI";   //Канал 4
               5:
                   #Signal := "Module12Chanel5_DI";   //Канал 5
               6:
                   #Signal := "Module12Chanel6_DI";   //Канал 6
               7:
                   #Signal := "Module12Chanel7_DI";   //Канал 7
               8:
                   #Signal := "Module12Chanel8_DI";   //Канал 8
               9:
                   #Signal := "Module12Chanel9_DI";   //Канал 9
               10:
                   #Signal := "Module12Chanel10_DI";  //Канал 10
               11:
                   #Signal := "Module12Chanel11_DI";  //Канал 11
               12:
                   #Signal := "Module12Chanel12_DI";  //Канал 12
               13:
                   #Signal := "Module12Chanel13_DI";  //Канал 13
               14:
                   #Signal := "Module12Chanel14_DI";  //Канал 14
               15:
                   #Signal := "Module12Chanel15_DI";  //Канал 15
               16:
                   #Signal := "Module12Chanel16_DI";  //Канал 16
               ELSE
                   #Signal := FALSE;
           END_CASE;
       13:  // Модуль 13
           CASE #N_chanel OF
               1:
                   #Signal := "Module13Chanel1_DI";   //Канал 1
               2:
                   #Signal := "Module13Chanel2_DI";   //Канал 2
               3:
                   #Signal := "Module13Chanel3_DI";   //Канал 3
               4:
                   #Signal := "Module13Chanel4_DI";   //Канал 4
               5:
                   #Signal := "Module13Chanel5_DI";   //Канал 5
               6:
                   #Signal := "Module13Chanel6_DI";   //Канал 6
               7:
                   #Signal := "Module13Chanel7_DI";   //Канал 7
               8:
                   #Signal := "Module13Chanel8_DI";   //Канал 8
               9:
                   #Signal := "Module13Chanel9_DI";   //Канал 9
               10:
                   #Signal := "Module13Chanel10_DI";  //Канал 10
               11:
                   #Signal := "Module13Chanel11_DI";  //Канал 11
               12:
                   #Signal := "Module13Chanel12_DI";  //Канал 12
               13:
                   #Signal := "Module13Chanel13_DI";  //Канал 13
               14:
                   #Signal := "Module13Chanel14_DI";  //Канал 14
               15:
                   #Signal := "Module13Chanel15_DI";  //Канал 15
               16:
                   #Signal := "Module13Chanel16_DI";  //Канал 16
               ELSE
                   #Signal := FALSE;
           END_CASE;
       14:  // Модуль 14
           CASE #N_chanel OF
               1:
                   #Signal := "Module14Chanel1_DI";   //Канал 1
               2:
                   #Signal := "Module14Chanel2_DI";   //Канал 2
               3:
                   #Signal := "Module14Chanel3_DI";   //Канал 3
               4:
                   #Signal := "Module14Chanel4_DI";   //Канал 4
               5:
                   #Signal := "Module14Chanel5_DI";   //Канал 5
               6:
                   #Signal := "Module14Chanel6_DI";   //Канал 6
               7:
                   #Signal := "Module14Chanel7_DI";   //Канал 7
               8:
                   #Signal := "Module14Chanel8_DI";   //Канал 8
               9:
                   #Signal := "Module14Chanel9_DI";   //Канал 9
               10:
                   #Signal := "Module14Chanel10_DI";  //Канал 10
               11:
                   #Signal := "Module14Chanel11_DI";  //Канал 11
               12:
                   #Signal := "Module14Chanel12_DI";  //Канал 12
               13:
                   #Signal := "Module14Chanel13_DI";  //Канал 13
               14:
                   #Signal := "Module14Chanel14_DI";  //Канал 14
               15:
                   #Signal := "Module14Chanel15_DI";  //Канал 15
               16:
                   #Signal := "Module14Chanel16_DI";  //Канал 16
               ELSE
                   #Signal := FALSE;
           END_CASE;
       15:  // Модуль 15
           CASE #N_chanel OF
               1:
                   #Signal := "Module15Chanel1_DI";   //Канал 1
               2:
                   #Signal := "Module15Chanel2_DI";   //Канал 2
               3:
                   #Signal := "Module15Chanel3_DI";   //Канал 3
               4:
                   #Signal := "Module15Chanel4_DI";   //Канал 4
               5:
                   #Signal := "Module15Chanel5_DI";   //Канал 5
               6:
                   #Signal := "Module15Chanel6_DI";   //Канал 6
               7:
                   #Signal := "Module15Chanel7_DI";   //Канал 7
               8:
                   #Signal := "Module15Chanel8_DI";   //Канал 8
               9:
                   #Signal := "Module15Chanel9_DI";   //Канал 9
               10:
                   #Signal := "Module15Chanel10_DI";  //Канал 10
               11:
                   #Signal := "Module15Chanel11_DI";  //Канал 11
               12:
                   #Signal := "Module15Chanel12_DI";  //Канал 12
               13:
                   #Signal := "Module15Chanel13_DI";  //Канал 13
               14:
                   #Signal := "Module15Chanel14_DI";  //Канал 14
               15:
                   #Signal := "Module15Chanel15_DI";  //Канал 15
               16:
                   #Signal := "Module15Chanel16_DI";  //Канал 16
               ELSE
                   #Signal := FALSE;
           END_CASE;
       16:  // Модуль 16
           CASE #N_chanel OF
               1:
                   #Signal := "Module16Chanel1_DI";   //Канал 1
               2:
                   #Signal := "Module16Chanel2_DI";   //Канал 2
               3:
                   #Signal := "Module16Chanel3_DI";   //Канал 3
               4:
                   #Signal := "Module16Chanel4_DI";   //Канал 4
               5:
                   #Signal := "Module16Chanel5_DI";   //Канал 5
               6:
                   #Signal := "Module16Chanel6_DI";   //Канал 6
               7:
                   #Signal := "Module16Chanel7_DI";   //Канал 7
               8:
                   #Signal := "Module16Chanel8_DI";   //Канал 8
               9:
                   #Signal := "Module16Chanel9_DI";   //Канал 9
               10:
                   #Signal := "Module16Chanel10_DI";  //Канал 10
               11:
                   #Signal := "Module16Chanel11_DI";  //Канал 11
               12:
                   #Signal := "Module16Chanel12_DI";  //Канал 12
               13:
                   #Signal := "Module16Chanel13_DI";  //Канал 13
               14:
                   #Signal := "Module16Chanel14_DI";  //Канал 14
               15:
                   #Signal := "Module16Chanel15_DI";  //Канал 15
               16:
                   #Signal := "Module16Chanel16_DI";  //Канал 16
               ELSE
                   #Signal := FALSE;
           END_CASE;
       17:  // Модуль 17
           CASE #N_chanel OF
               1:
                   #Signal := "Module17Chanel1_DI";   //Канал 1
               2:
                   #Signal := "Module17Chanel2_DI";   //Канал 2
               3:
                   #Signal := "Module17Chanel3_DI";   //Канал 3
               4:
                   #Signal := "Module17Chanel4_DI";   //Канал 4
               5:
                   #Signal := "Module17Chanel5_DI";   //Канал 5
               6:
                   #Signal := "Module17Chanel6_DI";   //Канал 6
               7:
                   #Signal := "Module17Chanel7_DI";   //Канал 7
               8:
                   #Signal := "Module17Chanel8_DI";   //Канал 8
               9:
                   #Signal := "Module17Chanel9_DI";   //Канал 9
               10:
                   #Signal := "Module17Chanel10_DI";  //Канал 10
               11:
                   #Signal := "Module17Chanel11_DI";  //Канал 11
               12:
                   #Signal := "Module17Chanel12_DI";  //Канал 12
               13:
                   #Signal := "Module17Chanel13_DI";  //Канал 13
               14:
                   #Signal := "Module17Chanel14_DI";  //Канал 14
               15:
                   #Signal := "Module17Chanel15_DI";  //Канал 15
               16:
                   #Signal := "Module17Chanel16_DI";  //Канал 16
               ELSE
                   #Signal := FALSE;
           END_CASE;
       18:  // Модуль 18
           CASE #N_chanel OF
               1:
                   #Signal := "Module18Chanel1_DI";   //Канал 1
               2:
                   #Signal := "Module18Chanel2_DI";   //Канал 2
               3:
                   #Signal := "Module18Chanel3_DI";   //Канал 3
               4:
                   #Signal := "Module18Chanel4_DI";   //Канал 4
               5:
                   #Signal := "Module18Chanel5_DI";   //Канал 5
               6:
                   #Signal := "Module18Chanel6_DI";   //Канал 6
               7:
                   #Signal := "Module18Chanel7_DI";   //Канал 7
               8:
                   #Signal := "Module18Chanel8_DI";   //Канал 8
               9:
                   #Signal := "Module18Chanel9_DI";   //Канал 9
               10:
                   #Signal := "Module18Chanel10_DI";  //Канал 10
               11:
                   #Signal := "Module18Chanel11_DI";  //Канал 11
               12:
                   #Signal := "Module18Chanel12_DI";  //Канал 12
               13:
                   #Signal := "Module18Chanel13_DI";  //Канал 13
               14:
                   #Signal := "Module18Chanel14_DI";  //Канал 14
               15:
                   #Signal := "Module18Chanel15_DI";  //Канал 15
               16:
                   #Signal := "Module18Chanel16_DI";  //Канал 16
               ELSE
                   #Signal := FALSE;
           END_CASE;
       19:  // Модуль 19
           CASE #N_chanel OF
               1:
                   #Signal := "Module19Chanel1_DI";   //Канал 1
               2:
                   #Signal := "Module19Chanel2_DI";   //Канал 2
               3:
                   #Signal := "Module19Chanel3_DI";   //Канал 3
               4:
                   #Signal := "Module19Chanel4_DI";   //Канал 4
               5:
                   #Signal := "Module19Chanel5_DI";   //Канал 5
               6:
                   #Signal := "Module19Chanel6_DI";   //Канал 6
               7:
                   #Signal := "Module19Chanel7_DI";   //Канал 7
               8:
                   #Signal := "Module19Chanel8_DI";   //Канал 8
               9:
                   #Signal := "Module19Chanel9_DI";   //Канал 9
               10:
                   #Signal := "Module19Chanel10_DI";  //Канал 10
               11:
                   #Signal := "Module19Chanel11_DI";  //Канал 11
               12:
                   #Signal := "Module19Chanel12_DI";  //Канал 12
               13:
                   #Signal := "Module19Chanel13_DI";  //Канал 13
               14:
                   #Signal := "Module19Chanel14_DI";  //Канал 14
               15:
                   #Signal := "Module19Chanel15_DI";  //Канал 15
               16:
                   #Signal := "Module19Chanel16_DI";  //Канал 16
               ELSE
                   #Signal := FALSE;
           END_CASE;
       20:  // Модуль 20
           CASE #N_chanel OF
               1:
                   #Signal := "Module20Chanel1_DI";   //Канал 1
               2:
                   #Signal := "Module20Chanel2_DI";   //Канал 2
               3:
                   #Signal := "Module20Chanel3_DI";   //Канал 3
               4:
                   #Signal := "Module20Chanel4_DI";   //Канал 4
               5:
                   #Signal := "Module20Chanel5_DI";   //Канал 5
               6:
                   #Signal := "Module20Chanel6_DI";   //Канал 6
               7:
                   #Signal := "Module20Chanel7_DI";   //Канал 7
               8:
                   #Signal := "Module20Chanel8_DI";   //Канал 8
               9:
                   #Signal := "Module20Chanel9_DI";   //Канал 9
               10:
                   #Signal := "Module20Chanel10_DI";  //Канал 10
               11:
                   #Signal := "Module20Chanel11_DI";  //Канал 11
               12:
                   #Signal := "Module20Chanel12_DI";  //Канал 12
               13:
                   #Signal := "Module20Chanel13_DI";  //Канал 13
               14:
                   #Signal := "Module20Chanel14_DI";  //Канал 14
               15:
                   #Signal := "Module20Chanel15_DI";  //Канал 15
               16:
                   #Signal := "Module20Chanel16_DI";  //Канал 16
               ELSE
                   #Signal := FALSE;
           END_CASE;
       21:  // Модуль 21
           CASE #N_chanel OF
               1:
                   #Signal := "Module21Chanel1_DI";   //Канал 1
               2:
                   #Signal := "Module21Chanel2_DI";   //Канал 2
               3:
                   #Signal := "Module21Chanel3_DI";   //Канал 3
               4:
                   #Signal := "Module21Chanel4_DI";   //Канал 4
               5:
                   #Signal := "Module21Chanel5_DI";   //Канал 5
               6:
                   #Signal := "Module21Chanel6_DI";   //Канал 6
               7:
                   #Signal := "Module21Chanel7_DI";   //Канал 7
               8:
                   #Signal := "Module21Chanel8_DI";   //Канал 8
               9:
                   #Signal := "Module21Chanel9_DI";   //Канал 9
               10:
                   #Signal := "Module21Chanel10_DI";  //Канал 10
               11:
                   #Signal := "Module21Chanel11_DI";  //Канал 11
               12:
                   #Signal := "Module21Chanel12_DI";  //Канал 12
               13:
                   #Signal := "Module21Chanel13_DI";  //Канал 13
               14:
                   #Signal := "Module21Chanel14_DI";  //Канал 14
               15:
                   #Signal := "Module21Chanel15_DI";  //Канал 15
               16:
                   #Signal := "Module21Chanel16_DI";  //Канал 16
               ELSE
                   #Signal := FALSE;
           END_CASE;
       22:  // Модуль 22
           CASE #N_chanel OF
               1:
                   #Signal := "Module22Chanel1_DI";   //Канал 1
               2:
                   #Signal := "Module22Chanel2_DI";   //Канал 2
               3:
                   #Signal := "Module22Chanel3_DI";   //Канал 3
               4:
                   #Signal := "Module22Chanel4_DI";   //Канал 4
               5:
                   #Signal := "Module22Chanel5_DI";   //Канал 5
               6:
                   #Signal := "Module22Chanel6_DI";   //Канал 6
               7:
                   #Signal := "Module22Chanel7_DI";   //Канал 7
               8:
                   #Signal := "Module22Chanel8_DI";   //Канал 8
               9:
                   #Signal := "Module22Chanel9_DI";   //Канал 9
               10:
                   #Signal := "Module22Chanel10_DI";  //Канал 10
               11:
                   #Signal := "Module22Chanel11_DI";  //Канал 11
               12:
                   #Signal := "Module22Chanel12_DI";  //Канал 12
               13:
                   #Signal := "Module22Chanel13_DI";  //Канал 13
               14:
                   #Signal := "Module22Chanel14_DI";  //Канал 14
               15:
                   #Signal := "Module22Chanel15_DI";  //Канал 15
               16:
                   #Signal := "Module22Chanel16_DI";  //Канал 16
               ELSE
                   #Signal := FALSE;
           END_CASE;
       23:  // Модуль 23
           CASE #N_chanel OF
               1:
                   #Signal := "Module23Chanel1_DI";   //Канал 1
               2:
                   #Signal := "Module23Chanel2_DI";   //Канал 2
               3:
                   #Signal := "Module23Chanel3_DI";   //Канал 3
               4:
                   #Signal := "Module23Chanel4_DI";   //Канал 4
               5:
                   #Signal := "Module23Chanel5_DI";   //Канал 5
               6:
                   #Signal := "Module23Chanel6_DI";   //Канал 6
               7:
                   #Signal := "Module23Chanel7_DI";   //Канал 7
               8:
                   #Signal := "Module23Chanel8_DI";   //Канал 8
               9:
                   #Signal := "Module23Chanel9_DI";   //Канал 9
               10:
                   #Signal := "Module23Chanel10_DI";  //Канал 10
               11:
                   #Signal := "Module23Chanel11_DI";  //Канал 11
               12:
                   #Signal := "Module23Chanel12_DI";  //Канал 12
               13:
                   #Signal := "Module23Chanel13_DI";  //Канал 13
               14:
                   #Signal := "Module23Chanel14_DI";  //Канал 14
               15:
                   #Signal := "Module23Chanel15_DI";  //Канал 15
               16:
                   #Signal := "Module23Chanel16_DI";  //Канал 16
               ELSE
                   #Signal := FALSE;
           END_CASE;
       24:  // Модуль 24
           CASE #N_chanel OF
               1:
                   #Signal := "Module24Chanel1_DI";   //Канал 1
               2:
                   #Signal := "Module24Chanel2_DI";   //Канал 2
               3:
                   #Signal := "Module24Chanel3_DI";   //Канал 3
               4:
                   #Signal := "Module24Chanel4_DI";   //Канал 4
               5:
                   #Signal := "Module24Chanel5_DI";   //Канал 5
               6:
                   #Signal := "Module24Chanel6_DI";   //Канал 6
               7:
                   #Signal := "Module24Chanel7_DI";   //Канал 7
               8:
                   #Signal := "Module24Chanel8_DI";   //Канал 8
               9:
                   #Signal := "Module24Chanel9_DI";   //Канал 9
               10:
                   #Signal := "Module24Chanel10_DI";  //Канал 10
               11:
                   #Signal := "Module24Chanel11_DI";  //Канал 11
               12:
                   #Signal := "Module24Chanel12_DI";  //Канал 12
               13:
                   #Signal := "Module24Chanel13_DI";  //Канал 13
               14:
                   #Signal := "Module24Chanel14_DI";  //Канал 14
               15:
                   #Signal := "Module24Chanel15_DI";  //Канал 15
               16:
                   #Signal := "Module24Chanel16_DI";  //Канал 16
               ELSE
                   #Signal := FALSE;
           END_CASE;
       25:  // Модуль 25
           CASE #N_chanel OF
               1:
                   #Signal := "Module25Chanel1_DI";   //Канал 1
               2:
                   #Signal := "Module25Chanel2_DI";   //Канал 2
               3:
                   #Signal := "Module25Chanel3_DI";   //Канал 3
               4:
                   #Signal := "Module25Chanel4_DI";   //Канал 4
               5:
                   #Signal := "Module25Chanel5_DI";   //Канал 5
               6:
                   #Signal := "Module25Chanel6_DI";   //Канал 6
               7:
                   #Signal := "Module25Chanel7_DI";   //Канал 7
               8:
                   #Signal := "Module25Chanel8_DI";   //Канал 8
               9:
                   #Signal := "Module25Chanel9_DI";   //Канал 9
               10:
                   #Signal := "Module25Chanel10_DI";  //Канал 10
               11:
                   #Signal := "Module25Chanel11_DI";  //Канал 11
               12:
                   #Signal := "Module25Chanel12_DI";  //Канал 12
               13:
                   #Signal := "Module25Chanel13_DI";  //Канал 13
               14:
                   #Signal := "Module25Chanel14_DI";  //Канал 14
               15:
                   #Signal := "Module25Chanel15_DI";  //Канал 15
               16:
                   #Signal := "Module25Chanel16_DI";  //Канал 16
               ELSE
                   #Signal := FALSE;
           END_CASE;
       ELSE
           #Signal := FALSE;
   END_CASE;
   IF NOT #Invert THEN
       #read_discret:= #Signal;
   ELSE
       #read_discret:= NOT #Signal;
   END_IF;
END_FUNCTION

FUNCTION "read_4_20" : Real   // FC3, SCL
{ S7_Optimized_Access := 'TRUE' }
AUTHOR : Dmitriy_Petrov
VERSION : 0.1
// Функция чтения сигнала 4-20mA
   VAR_INPUT
      LL_sensor : Real;   // Нижний предел датчика в физической величине
      HL_sensor : Real;   // Верхний предел датчика в физической величине
      LL_ADC : Int;   // Нижний предел АЦП
      HL_ADC : Int;   // Верхний предел АЦП
   END_VAR
   VAR_OUTPUT
      Current : Real;   // Значение тока
      error_sensor : Bool;   // Неисправность датчика
   END_VAR
   VAR_IN_OUT
      N_module : USInt;   // № модуля (начиная с 1)
      N_chanel : USInt;   // № канала (начиная с 1)
      ADC : Int;   // Текущий код АЦП
   END_VAR
   VAR_TEMP
      K : Real;   // Коэффициент К
      "B" : Real;   // Коэффициент B
   END_VAR
BEGIN
   (*проверка правильности введенного значения № Модуля*)
   IF #N_module < 1 OR #N_module > 25 THEN
       #N_module := 0;
   END_IF;

   (*проверка правильности введенного значения № Канала*)
   IF #N_module = 0 THEN
       #N_chanel := 0;
   ELSE
       IF #N_chanel < 1 OR #N_chanel > 8 THEN
           #N_chanel := 0;
       END_IF;
   END_IF;

   (*считывание кода АЦП выбранного канала*)
   CASE #N_module OF
       1:  // Модуль 1
           CASE #N_chanel OF
               1:
                   #ADC := "Module01Chanel1_AI";   //Канал 1
               2:
                   #ADC := "Module01Chanel2_AI";   //Канал 2
               3:
                   #ADC := "Module01Chanel3_AI";   //Канал 3
               4:
                   #ADC := "Module01Chanel4_AI";   //Канал 4
               5:
                   #ADC := "Module01Chanel5_AI";   //Канал 5
               6:
                   #ADC := "Module01Chanel6_AI";   //Канал 6
               7:
                   #ADC := "Module01Chanel7_AI";   //Канал 7
               8:
                   #ADC := "Module01Chanel8_AI";   //Канал 8
               ELSE
                   #ADC := 0;
           END_CASE;
       2:  // Модуль 2
           CASE #N_chanel OF
               1:
                   #ADC := "Module02Chanel1_AI";   //Канал 1
               2:
                   #ADC := "Module02Chanel2_AI";   //Канал 2
               3:
                   #ADC := "Module02Chanel3_AI";   //Канал 3
               4:
                   #ADC := "Module02Chanel4_AI";   //Канал 4
               5:
                   #ADC := "Module02Chanel5_AI";   //Канал 5
               6:
                   #ADC := "Module02Chanel6_AI";   //Канал 6
               7:
                   #ADC := "Module02Chanel7_AI";   //Канал 7
               8:
                   #ADC := "Module02Chanel8_AI";   //Канал 8
               ELSE
                   #ADC := 0;
           END_CASE;
       3:  // Модуль 3
           CASE #N_chanel OF
               1:
                   #ADC := "Module03Chanel1_AI";   //Канал 1
               2:
                   #ADC := "Module03Chanel2_AI";   //Канал 2
               3:
                   #ADC := "Module03Chanel3_AI";   //Канал 3
               4:
                   #ADC := "Module03Chanel4_AI";   //Канал 4
               5:
                   #ADC := "Module03Chanel5_AI";   //Канал 5
               6:
                   #ADC := "Module03Chanel6_AI";   //Канал 6
               7:
                   #ADC := "Module03Chanel7_AI";   //Канал 7
               8:
                   #ADC := "Module03Chanel8_AI";   //Канал 8
               ELSE
                   #ADC := 0;
           END_CASE;
       4:  // Модуль 4
           CASE #N_chanel OF
               1:
                   #ADC := "Module04Chanel1_AI";   //Канал 1
               2:
                   #ADC := "Module04Chanel2_AI";   //Канал 2
               3:
                   #ADC := "Module04Chanel3_AI";   //Канал 3
               4:
                   #ADC := "Module04Chanel4_AI";   //Канал 4
               5:
                   #ADC := "Module04Chanel5_AI";   //Канал 5
               6:
                   #ADC := "Module04Chanel6_AI";   //Канал 6
               7:
                   #ADC := "Module04Chanel7_AI";   //Канал 7
               8:
                   #ADC := "Module04Chanel8_AI";   //Канал 8
               ELSE
                   #ADC := 0;
           END_CASE;
       5:  // Модуль 5
           CASE #N_chanel OF
               1:
                   #ADC := "Module05Chanel1_AI";   //Канал 1
               2:
                   #ADC := "Module05Chanel2_AI";   //Канал 2
               3:
                   #ADC := "Module05Chanel3_AI";   //Канал 3
               4:
                   #ADC := "Module05Chanel4_AI";   //Канал 4
               5:
                   #ADC := "Module05Chanel5_AI";   //Канал 5
               6:
                   #ADC := "Module05Chanel6_AI";   //Канал 6
               7:
                   #ADC := "Module05Chanel7_AI";   //Канал 7
               8:
                   #ADC := "Module05Chanel8_AI";   //Канал 8
               ELSE
                   #ADC := 0;
           END_CASE;
       6:  // Модуль 6
           CASE #N_chanel OF
               1:
                   #ADC := "Module06Chanel1_AI";   //Канал 1
               2:
                   #ADC := "Module06Chanel2_AI";   //Канал 2
               3:
                   #ADC := "Module06Chanel3_AI";   //Канал 3
               4:
                   #ADC := "Module06Chanel4_AI";   //Канал 4
               5:
                   #ADC := "Module06Chanel5_AI";   //Канал 5
               6:
                   #ADC := "Module06Chanel6_AI";   //Канал 6
               7:
                   #ADC := "Module06Chanel7_AI";   //Канал 7
               8:
                   #ADC := "Module06Chanel8_AI";   //Канал 8
               ELSE
                   #ADC := 0;
           END_CASE;
       7:  // Модуль 7
           CASE #N_chanel OF
               1:
                   #ADC := "Module07Chanel1_AI";   //Канал 1
               2:
                   #ADC := "Module07Chanel2_AI";   //Канал 2
               3:
                   #ADC := "Module07Chanel3_AI";   //Канал 3
               4:
                   #ADC := "Module07Chanel4_AI";   //Канал 4
               5:
                   #ADC := "Module07Chanel5_AI";   //Канал 5
               6:
                   #ADC := "Module07Chanel6_AI";   //Канал 6
               7:
                   #ADC := "Module07Chanel7_AI";   //Канал 7
               8:
                   #ADC := "Module07Chanel8_AI";   //Канал 8
               ELSE
                   #ADC := 0;
           END_CASE;
       8:  // Модуль 8
           CASE #N_chanel OF
               1:
                   #ADC := "Module08Chanel1_AI";   //Канал 1
               2:
                   #ADC := "Module08Chanel2_AI";   //Канал 2
               3:
                   #ADC := "Module08Chanel3_AI";   //Канал 3
               4:
                   #ADC := "Module08Chanel4_AI";   //Канал 4
               5:
                   #ADC := "Module08Chanel5_AI";   //Канал 5
               6:
                   #ADC := "Module08Chanel6_AI";   //Канал 6
               7:
                   #ADC := "Module08Chanel7_AI";   //Канал 7
               8:
                   #ADC := "Module08Chanel8_AI";   //Канал 8
               ELSE
                   #ADC := 0;
           END_CASE;
       9:  // Модуль 9
           CASE #N_chanel OF
               1:
                   #ADC := "Module09Chanel1_AI";   //Канал 1
               2:
                   #ADC := "Module09Chanel2_AI";   //Канал 2
               3:
                   #ADC := "Module09Chanel3_AI";   //Канал 3
               4:
                   #ADC := "Module09Chanel4_AI";   //Канал 4
               5:
                   #ADC := "Module09Chanel5_AI";   //Канал 5
               6:
                   #ADC := "Module09Chanel6_AI";   //Канал 6
               7:
                   #ADC := "Module09Chanel7_AI";   //Канал 7
               8:
                   #ADC := "Module09Chanel8_AI";   //Канал 8
               ELSE
                   #ADC := 0;
           END_CASE;
       10:  // Модуль 10
           CASE #N_chanel OF
               1:
                   #ADC := "Module10Chanel1_AI";   //Канал 1
               2:
                   #ADC := "Module10Chanel2_AI";   //Канал 2
               3:
                   #ADC := "Module10Chanel3_AI";   //Канал 3
               4:
                   #ADC := "Module10Chanel4_AI";   //Канал 4
               5:
                   #ADC := "Module10Chanel5_AI";   //Канал 5
               6:
                   #ADC := "Module10Chanel6_AI";   //Канал 6
               7:
                   #ADC := "Module10Chanel7_AI";   //Канал 7
               8:
                   #ADC := "Module10Chanel8_AI";   //Канал 8
               ELSE
                   #ADC := 0;
           END_CASE;
       11:  // Модуль 11
           CASE #N_chanel OF
               1:
                   #ADC := "Module11Chanel1_AI";   //Канал 1
               2:
                   #ADC := "Module11Chanel2_AI";   //Канал 2
               3:
                   #ADC := "Module11Chanel3_AI";   //Канал 3
               4:
                   #ADC := "Module11Chanel4_AI";   //Канал 4
               5:
                   #ADC := "Module11Chanel5_AI";   //Канал 5
               6:
                   #ADC := "Module11Chanel6_AI";   //Канал 6
               7:
                   #ADC := "Module11Chanel7_AI";   //Канал 7
               8:
                   #ADC := "Module11Chanel8_AI";   //Канал 8
               ELSE
                   #ADC := 0;
           END_CASE;
       12:  // Модуль 12
           CASE #N_chanel OF
               1:
                   #ADC := "Module12Chanel1_AI";   //Канал 1
               2:
                   #ADC := "Module12Chanel2_AI";   //Канал 2
               3:
                   #ADC := "Module12Chanel3_AI";   //Канал 3
               4:
                   #ADC := "Module12Chanel4_AI";   //Канал 4
               5:
                   #ADC := "Module12Chanel5_AI";   //Канал 5
               6:
                   #ADC := "Module12Chanel6_AI";   //Канал 6
               7:
                   #ADC := "Module12Chanel7_AI";   //Канал 7
               8:
                   #ADC := "Module12Chanel8_AI";   //Канал 8
               ELSE
                   #ADC := 0;
           END_CASE;
       13:  // Модуль 13
           CASE #N_chanel OF
               1:
                   #ADC := "Module13Chanel1_AI";   //Канал 1
               2:
                   #ADC := "Module13Chanel2_AI";   //Канал 2
               3:
                   #ADC := "Module13Chanel3_AI";   //Канал 3
               4:
                   #ADC := "Module13Chanel4_AI";   //Канал 4
               5:
                   #ADC := "Module13Chanel5_AI";   //Канал 5
               6:
                   #ADC := "Module13Chanel6_AI";   //Канал 6
               7:
                   #ADC := "Module13Chanel7_AI";   //Канал 7
               8:
                   #ADC := "Module13Chanel8_AI";   //Канал 8
               ELSE
                   #ADC := 0;
           END_CASE;
       14:  // Модуль 14
           CASE #N_chanel OF
               1:
                   #ADC := "Module14Chanel1_AI";   //Канал 1
               2:
                   #ADC := "Module14Chanel2_AI";   //Канал 2
               3:
                   #ADC := "Module14Chanel3_AI";   //Канал 3
               4:
                   #ADC := "Module14Chanel4_AI";   //Канал 4
               5:
                   #ADC := "Module14Chanel5_AI";   //Канал 5
               6:
                   #ADC := "Module14Chanel6_AI";   //Канал 6
               7:
                   #ADC := "Module14Chanel7_AI";   //Канал 7
               8:
                   #ADC := "Module14Chanel8_AI";   //Канал 8
               ELSE
                   #ADC := 0;
           END_CASE;
       15:  // Модуль 15
           CASE #N_chanel OF
               1:
                   #ADC := "Module15Chanel1_AI";   //Канал 1
               2:
                   #ADC := "Module15Chanel2_AI";   //Канал 2
               3:
                   #ADC := "Module15Chanel3_AI";   //Канал 3
               4:
                   #ADC := "Module15Chanel4_AI";   //Канал 4
               5:
                   #ADC := "Module15Chanel5_AI";   //Канал 5
               6:
                   #ADC := "Module15Chanel6_AI";   //Канал 6
               7:
                   #ADC := "Module15Chanel7_AI";   //Канал 7
               8:
                   #ADC := "Module15Chanel8_AI";   //Канал 8
               ELSE
                   #ADC := 0;
           END_CASE;
       16:  // Модуль 16
           CASE #N_chanel OF
               1:
                   #ADC := "Module16Chanel1_AI";   //Канал 1
               2:
                   #ADC := "Module16Chanel2_AI";   //Канал 2
               3:
                   #ADC := "Module16Chanel3_AI";   //Канал 3
               4:
                   #ADC := "Module16Chanel4_AI";   //Канал 4
               5:
                   #ADC := "Module16Chanel5_AI";   //Канал 5
               6:
                   #ADC := "Module16Chanel6_AI";   //Канал 6
               7:
                   #ADC := "Module16Chanel7_AI";   //Канал 7
               8:
                   #ADC := "Module16Chanel8_AI";   //Канал 8
               ELSE
                   #ADC := 0;
           END_CASE;
       17:  // Модуль 17
           CASE #N_chanel OF
               1:
                   #ADC := "Module17Chanel1_AI";   //Канал 1
               2:
                   #ADC := "Module17Chanel2_AI";   //Канал 2
               3:
                   #ADC := "Module17Chanel3_AI";   //Канал 3
               4:
                   #ADC := "Module17Chanel4_AI";   //Канал 4
               5:
                   #ADC := "Module17Chanel5_AI";   //Канал 5
               6:
                   #ADC := "Module17Chanel6_AI";   //Канал 6
               7:
                   #ADC := "Module17Chanel7_AI";   //Канал 7
               8:
                   #ADC := "Module17Chanel8_AI";   //Канал 8
               ELSE
                   #ADC := 0;
           END_CASE;
       18:  // Модуль 18
           CASE #N_chanel OF
               1:
                   #ADC := "Module18Chanel1_AI";   //Канал 1
               2:
                   #ADC := "Module18Chanel2_AI";   //Канал 2
               3:
                   #ADC := "Module18Chanel3_AI";   //Канал 3
               4:
                   #ADC := "Module18Chanel4_AI";   //Канал 4
               5:
                   #ADC := "Module18Chanel5_AI";   //Канал 5
               6:
                   #ADC := "Module18Chanel6_AI";   //Канал 6
               7:
                   #ADC := "Module18Chanel7_AI";   //Канал 7
               8:
                   #ADC := "Module18Chanel8_AI";   //Канал 8
               ELSE
                   #ADC := 0;
           END_CASE;
       19:  // Модуль 19
           CASE #N_chanel OF
               1:
                   #ADC := "Module19Chanel1_AI";   //Канал 1
               2:
                   #ADC := "Module19Chanel2_AI";   //Канал 2
               3:
                   #ADC := "Module19Chanel3_AI";   //Канал 3
               4:
                   #ADC := "Module19Chanel4_AI";   //Канал 4
               5:
                   #ADC := "Module19Chanel5_AI";   //Канал 5
               6:
                   #ADC := "Module19Chanel6_AI";   //Канал 6
               7:
                   #ADC := "Module19Chanel7_AI";   //Канал 7
               8:
                   #ADC := "Module19Chanel8_AI";   //Канал 8
               ELSE
                   #ADC := 0;
           END_CASE;
       20:  // Модуль 20
           CASE #N_chanel OF
               1:
                   #ADC := "Module20Chanel1_AI";   //Канал 1
               2:
                   #ADC := "Module20Chanel2_AI";   //Канал 2
               3:
                   #ADC := "Module20Chanel3_AI";   //Канал 3
               4:
                   #ADC := "Module20Chanel4_AI";   //Канал 4
               5:
                   #ADC := "Module20Chanel5_AI";   //Канал 5
               6:
                   #ADC := "Module20Chanel6_AI";   //Канал 6
               7:
                   #ADC := "Module20Chanel7_AI";   //Канал 7
               8:
                   #ADC := "Module20Chanel8_AI";   //Канал 8
               ELSE
                   #ADC := 0;
           END_CASE;
       21:  // Модуль 21
           CASE #N_chanel OF
               1:
                   #ADC := "Module21Chanel1_AI";   //Канал 1
               2:
                   #ADC := "Module21Chanel2_AI";   //Канал 2
               3:
                   #ADC := "Module21Chanel3_AI";   //Канал 3
               4:
                   #ADC := "Module21Chanel4_AI";   //Канал 4
               5:
                   #ADC := "Module21Chanel5_AI";   //Канал 5
               6:
                   #ADC := "Module21Chanel6_AI";   //Канал 6
               7:
                   #ADC := "Module21Chanel7_AI";   //Канал 7
               8:
                   #ADC := "Module21Chanel8_AI";   //Канал 8
               ELSE
                   #ADC := 0;
           END_CASE;
       22:  // Модуль 22
           CASE #N_chanel OF
               1:
                   #ADC := "Module22Chanel1_AI";   //Канал 1
               2:
                   #ADC := "Module22Chanel2_AI";   //Канал 2
               3:
                   #ADC := "Module22Chanel3_AI";   //Канал 3
               4:
                   #ADC := "Module22Chanel4_AI";   //Канал 4
               5:
                   #ADC := "Module22Chanel5_AI";   //Канал 5
               6:
                   #ADC := "Module22Chanel6_AI";   //Канал 6
               7:
                   #ADC := "Module22Chanel7_AI";   //Канал 7
               8:
                   #ADC := "Module22Chanel8_AI";   //Канал 8
               ELSE
                   #ADC := 0;
           END_CASE;
       23:  // Модуль 23
           CASE #N_chanel OF
               1:
                   #ADC := "Module23Chanel1_AI";   //Канал 1
               2:
                   #ADC := "Module23Chanel2_AI";   //Канал 2
               3:
                   #ADC := "Module23Chanel3_AI";   //Канал 3
               4:
                   #ADC := "Module23Chanel4_AI";   //Канал 4
               5:
                   #ADC := "Module23Chanel5_AI";   //Канал 5
               6:
                   #ADC := "Module23Chanel6_AI";   //Канал 6
               7:
                   #ADC := "Module23Chanel7_AI";   //Канал 7
               8:
                   #ADC := "Module23Chanel8_AI";   //Канал 8
               ELSE
                   #ADC := 0;
           END_CASE;
       24:  // Модуль 24
           CASE #N_chanel OF
               1:
                   #ADC := "Module24Chanel1_AI";   //Канал 1
               2:
                   #ADC := "Module24Chanel2_AI";   //Канал 2
               3:
                   #ADC := "Module24Chanel3_AI";   //Канал 3
               4:
                   #ADC := "Module24Chanel4_AI";   //Канал 4
               5:
                   #ADC := "Module24Chanel5_AI";   //Канал 5
               6:
                   #ADC := "Module24Chanel6_AI";   //Канал 6
               7:
                   #ADC := "Module24Chanel7_AI";   //Канал 7
               8:
                   #ADC := "Module24Chanel8_AI";   //Канал 8
               ELSE
                   #ADC := 0;
           END_CASE;
       25:  // Модуль 25
           CASE #N_chanel OF
               1:
                   #ADC := "Module25Chanel1_AI";   //Канал 1
               2:
                   #ADC := "Module25Chanel2_AI";   //Канал 2
               3:
                   #ADC := "Module25Chanel3_AI";   //Канал 3
               4:
                   #ADC := "Module25Chanel4_AI";   //Канал 4
               5:
                   #ADC := "Module25Chanel5_AI";   //Канал 5
               6:
                   #ADC := "Module25Chanel6_AI";   //Канал 6
               7:
                   #ADC := "Module25Chanel7_AI";   //Канал 7
               8:
                   #ADC := "Module25Chanel8_AI";   //Канал 8
               ELSE
                   #ADC := 0;
           END_CASE;
       ELSE
           #ADC := 0;
   END_CASE;

   (*вычисление физического значения*)
   #K := (#HL_sensor - #LL_sensor) / (#HL_ADC - #LL_ADC);
   #"B" := #LL_sensor - (#K * #LL_ADC);

   IF #ADC >= -4864 AND #ADC <= 32511 THEN
       #read_4_20 := (#K * #ADC) + #"B";
       #error_sensor := false;
   ELSE
       #error_sensor := true;
       IF #ADC < -4864 THEN
           #read_4_20 := -99999;
       ELSE
           #read_4_20 := 99999;
       END_IF;
   END_IF;

   (*вычисление физического значения тока*)
   #Current := (((20 - 4) / (INT_TO_REAL(27648 - 0))) * (INT_TO_REAL(#ADC))) + 4;
END_FUNCTION

FUNCTION "Write_outputs" : Void   // FC4, SCL
{ S7_Optimized_Access := 'TRUE' }
VERSION : 0.1
BEGIN
   (*ЗАПИСЬ ВЫХОДОВ*)
   (*Запись дискретных выходов*)
   //ЗРГ Команда «Больше»
   "ZRG_control_open"();
   //ЗРГ Команда «Меньше»
   "ZRG_control_close"();
   //НАВ Команда «Больше»
   "NAV_control_open"();
   //НАВ Команда «Меньше»
   "NAV_control_close"();
   //НАД Команда «Больше»
   "NAD_control_open"();
   //НАД Команда «Меньше»
   "NAD_control_close"();
   //ЗРВ Команда «Больше»
   "ZRW_control_open"();
   //ЗРВ Команда «Меньше»
   "ZRW_control_close"();
   //Индикация «Работа»
   "Indication_RUN"();
   //Индикация «Авария»
   "Indication_ALARM"();
   //Индикация «Защиты в норме»
   "Indication_NORMA"();
   //Индикация «Готов к розжигу»
   "Indication_READY"();

   (*Команда «Больше» управления мощностью резервной горелки

   Команда «Меньше» управления мощностью резервной горелки

   Команда «Ограничение мощности резервной горелки»*)

   //ЗДГ команда «открыть»
   "ZDG_control_open"();
   //ЗДГ команда «закрыть»
   "ZDG_control_close"();
   //ЗДГ команда «стоп»
   "ZDG_control_stop"();
   //ЗДГ команда «запрет открытия»
   "ZDG_control_disable_open"();
   //КБ команда «закрыть»
   "KB_control_close"();
   //КО команда «открыть»
   "KO_control_open"();
   //КЗ команда «открыть»
   "KZ_control_open"();
   //ИВН команда «включить»
   "IVN_control_on"();
   //ПЗК1 команда «открыть»
   "PZK1_control_open"();
   //ПЗК2 команда «открыть»
   "PZK2_control_open"();
   //ЗДСВ перед котлом команда «открыть»
   "ZDSV_before_boiler_control_open"();
   //ЗДСВ перед котлом команда «закрыть»
   "ZDSV_before_boiler_control_close"();
   //ЗДСВ перед котлом команда «стоп»
   "ZDSV_before_boiler_control_stop"();
   //ЗДСВ перед котлом команда «разрешение на закрытие»
   "ZDSV_before_boiler_control_disable_close"();
   //ГПЗ команда «открыть»
   "GPZ_control_open"();
   //ГПЗ команда «закрыть»
   "GPZ_control_close"();
   //ГПЗ команда «стоп»
   "GPZ_control_stop"();
   //ГПЗ команда «разрешение на закрытие»
   "GPZ_control_disable_close"();
   //Включение аварийной сигнализации
   "control_alarm_signal"();
   //ДВ команда «пуск»
   "DV_control_start"();
   //ДВ команда «стоп»
   "DV_control_stop"();
   //ДС команда «пуск»
   "DS_control_start"();
   //ДС команда «стоп»
   "DS_control_stop"();

   (*Запись аналоговых выходов*)
   //Задание для ПЧ ДВ
   "DV_control_frequency"();
   //Задание для ПЧ ДС
   "DS_control_frequency"();
END_FUNCTION

FUNCTION "Alarms_and_warnings" : Void   // FC5, SCL
{ S7_Optimized_Access := 'TRUE' }
VERSION : 0.1
BEGIN
   (*АВАРИИ*)
   "TON_alarm_1_DB".TON(IN := "Alarm_Timer".alarm_1_IN,
                        PT := "Alarm_Timer".alarm_1_PT,
                        Q => "Alarm_Timer".alarm_1_Q);
   "TON_alarm_2_DB".TON(IN := "Alarm_Timer".alarm_2_IN,
                        PT := "Alarm_Timer".alarm_2_PT,
                        Q => "Alarm_Timer".alarm_2_Q);
   "TON_alarm_3_DB".TON(IN := "Alarm_Timer".alarm_3_IN,
                        PT := "Alarm_Timer".alarm_3_PT,
                        Q => "Alarm_Timer".alarm_3_Q);
   "TON_alarm_4_DB".TON(IN := "Alarm_Timer".alarm_4_IN,
                        PT := "Alarm_Timer".alarm_4_PT,
                        Q => "Alarm_Timer".alarm_4_Q);
   "TON_alarm_5_DB".TON(IN := "Alarm_Timer".alarm_5_IN,
                        PT := "Alarm_Timer".alarm_5_PT,
                        Q => "Alarm_Timer".alarm_5_Q);
   "TON_alarm_6_DB".TON(IN := "Alarm_Timer".alarm_6_IN,
                        PT := "Alarm_Timer".alarm_6_PT,
                        Q => "Alarm_Timer".alarm_6_Q);
   "TON_alarm_7_DB".TON(IN := "Alarm_Timer".alarm_7_IN,
                        PT := "Alarm_Timer".alarm_7_PT,
                        Q => "Alarm_Timer".alarm_7_Q);
   "TON_alarm_8_DB".TON(IN := "Alarm_Timer".alarm_8_IN,
                        PT := "Alarm_Timer".alarm_8_PT,
                        Q => "Alarm_Timer".alarm_8_Q);
   "TON_alarm_9_DB".TON(IN := "Alarm_Timer".alarm_9_IN,
                        PT := "Alarm_Timer".alarm_9_PT,
                        Q => "Alarm_Timer".alarm_9_Q);
   "TON_alarm_10_DB".TON(IN := "Alarm_Timer".alarm_10_IN,
                        PT := "Alarm_Timer".alarm_10_PT,
                        Q => "Alarm_Timer".alarm_10_Q);
   "TON_alarm_11_DB".TON(IN := "Alarm_Timer".alarm_11_IN,
                        PT := "Alarm_Timer".alarm_11_PT,
                        Q => "Alarm_Timer".alarm_11_Q);
   "TON_alarm_12_DB".TON(IN := "Alarm_Timer".alarm_12_IN,
                        PT := "Alarm_Timer".alarm_12_PT,
                        Q => "Alarm_Timer".alarm_12_Q);
   "TON_alarm_13_DB".TON(IN := "Alarm_Timer".alarm_13_IN,
                        PT := "Alarm_Timer".alarm_13_PT,
                        Q => "Alarm_Timer".alarm_13_Q);
   "TON_alarm_14_DB".TON(IN := "Alarm_Timer".alarm_14_IN,
                        PT := "Alarm_Timer".alarm_14_PT,
                        Q => "Alarm_Timer".alarm_14_Q);
   "TON_alarm_15_DB".TON(IN := "Alarm_Timer".alarm_15_IN,
                        PT := "Alarm_Timer".alarm_15_PT,
                        Q => "Alarm_Timer".alarm_15_Q);
   "TON_alarm_16_DB".TON(IN := "Alarm_Timer".alarm_16_IN,
                        PT := "Alarm_Timer".alarm_16_PT,
                        Q => "Alarm_Timer".alarm_16_Q);
   "TON_alarm_17_DB".TON(IN := "Alarm_Timer".alarm_17_IN,
                        PT := "Alarm_Timer".alarm_17_PT,
                        Q => "Alarm_Timer".alarm_17_Q);

   (*Повышение давления газа перед БГ*)
   "Alarm_Timer".alarm_1_PT := T_CONV(INT_TO_DINT("Alarm_SP".TIME_P_gas_before_BG_max) * 1000);
   IF "Alarm_Enable".P_gas_before_BG_max THEN
       "Alarm_Timer".alarm_1_IN := "P_gas_before_BG_max".Value OR ("P_gas_before_BG".Value > "Alarm_SP".P_gas_before_BG_max AND NOT "P_gas_before_BG".Error_sensor AND "P_gas_before_BG".N_module<>0);
       IF "Alarm_Timer".alarm_1_Q THEN
           "Alarm".P_gas_before_BG_max := TRUE;
       END_IF;
   ELSE
       "Alarm_Timer".alarm_1_IN := FALSE;
   END_IF;
   //Формирование технологической защиты. Повышение давления газа перед БГ
   IF NOT "Protections_BLOCK".P_gas_before_BG_max THEN
       "Protections".P_gas_before_BG_max := "Alarm_Timer".alarm_1_Q;
   ELSE
       "Protections".P_gas_before_BG_max := FALSE;
   END_IF;

   (*Понижение давления газа перед БГ*)
   "Alarm_Timer".alarm_2_PT := T_CONV(INT_TO_DINT("Alarm_SP".TIME_P_gas_before_BG_min) * 1000);
   IF "Alarm_Enable".P_gas_before_BG_min THEN
       "Alarm_Timer".alarm_2_IN := "P_gas_before_BG_min".Value OR ("P_gas_before_BG".Value < "Alarm_SP".P_gas_before_BG_min AND NOT "P_gas_before_BG".Error_sensor AND "P_gas_before_BG".N_module<>0);
       IF "Alarm_Timer".alarm_2_Q THEN
           "Alarm".P_gas_before_BG_min := TRUE;
       END_IF;
   ELSE
       "Alarm_Timer".alarm_2_IN := FALSE;
   END_IF;
   //Формирование технологической защиты. Понижение давления газа перед БГ
   IF NOT "Protections_BLOCK".P_gas_before_BG_min THEN
       "Protections".P_gas_before_BG_min := "Alarm_Timer".alarm_2_Q;
   ELSE
       "Protections".P_gas_before_BG_min := FALSE;
   END_IF;

   (*Понижение давления газа перед горелкой*)
   "Alarm_Timer".alarm_3_PT := T_CONV(INT_TO_DINT("Alarm_SP".TIME_P_gas_before_burner_min) * 1000);
   IF "Alarm_Enable".P_gas_before_burner_min THEN
       "Alarm_Timer".alarm_3_IN := "P_gas_before_burner_min".Value OR ("P_gas_before_burner".Value < "Alarm_SP".P_gas_before_burner_min AND NOT "P_gas_before_burner".Error_sensor AND "P_gas_before_burner".N_module<>0);
       IF "Alarm_Timer".alarm_3_Q THEN
           "Alarm".P_gas_before_burner_min := TRUE;
       END_IF;
   ELSE
       "Alarm_Timer".alarm_3_IN := FALSE;
   END_IF;
   //Формирование технологической защиты. Понижение давления газа перед горелкой
   IF NOT "Protections_BLOCK".P_gas_before_burner_min THEN
       "Protections".P_gas_before_burner_min := "Alarm_Timer".alarm_3_Q;
   ELSE
       "Protections".P_gas_before_burner_min := FALSE;
   END_IF;

   (*Повышение давления газа перед горелкой*)
   "Alarm_Timer".alarm_4_PT := T_CONV(INT_TO_DINT("Alarm_SP".TIME_P_gas_before_burner_max) * 1000);
   IF "Alarm_Enable".P_gas_before_burner_max THEN
       "Alarm_Timer".alarm_4_IN := "P_gas_before_burner_max".Value OR ("P_gas_before_burner".Value > "Alarm_SP".P_gas_before_burner_max AND NOT "P_gas_before_burner".Error_sensor AND "P_gas_before_burner".N_module<>0);
       IF "Alarm_Timer".alarm_4_Q THEN
           "Alarm".P_gas_before_burner_max := TRUE;
       END_IF;
   ELSE
       "Alarm_Timer".alarm_4_IN := FALSE;
   END_IF;
   //Формирование технологической защиты. Повышение давления газа перед горелкой
   IF NOT "Protections_BLOCK".P_gas_before_burner_max THEN
       "Protections".P_gas_before_burner_max := "Alarm_Timer".alarm_4_Q;
   ELSE
       "Protections".P_gas_before_burner_max := FALSE;
   END_IF;

   (*Отключение ДС*)
   "Alarm_Timer".alarm_5_PT := T_CONV(INT_TO_DINT("Alarm_SP".TIME_DS_off) * 1000);
   IF "Alarm_Enable".DS_off THEN
       "Alarm_Timer".alarm_5_IN := (NOT "DS_invertor_on".Value AND NOT "DS_powergrid_on".Value);
       IF "Alarm_Timer".alarm_5_Q THEN
           "Alarm".DS_off := TRUE;
       END_IF;
   ELSE
       "Alarm_Timer".alarm_5_IN := FALSE;
   END_IF;
   //Формирование технологической защиты. Отключение ДС
   IF NOT "Protections_BLOCK".DS_off THEN
       "Protections".DS_off := "Alarm_Timer".alarm_5_Q;
   ELSE
       "Protections".DS_off := FALSE;
   END_IF;

   (*Отключение ДВ*)
   "Alarm_Timer".alarm_6_PT := T_CONV(INT_TO_DINT("Alarm_SP".TIME_DV_off) * 1000);
   IF "Alarm_Enable".DV_off THEN
       "Alarm_Timer".alarm_6_IN := (NOT "DV_invertor_on".Value AND NOT "DV_powergrid_on".Value);
       IF "Alarm_Timer".alarm_6_Q THEN
           "Alarm".DV_off := TRUE;
       END_IF;
   ELSE
       "Alarm_Timer".alarm_6_IN := FALSE;
   END_IF;
   //Формирование технологической защиты. Отключение ДВ
   IF NOT "Protections_BLOCK".DV_off THEN
       "Protections".DV_off := "Alarm_Timer".alarm_6_Q;
   ELSE
       "Protections".DV_off := FALSE;
   END_IF;

   (*Понижение разряжения в топке*)
   "Alarm_Timer".alarm_7_PT := T_CONV(INT_TO_DINT("Alarm_SP".TIME_dP_furnace_boiler_min) * 1000);
   IF "Alarm_Enable".dP_furnace_boiler_min THEN
       "Alarm_Timer".alarm_7_IN := "dP_furnace_boiler_min".Value OR ("dP_furnace_boiler".Value > "Alarm_SP".dP_furnace_boiler_min AND NOT "dP_furnace_boiler".Error_sensor AND "dP_furnace_boiler".N_module<>0);
       IF "Alarm_Timer".alarm_7_Q THEN
           "Alarm".dP_furnace_boiler_min := TRUE;
       END_IF;
   ELSE
       "Alarm_Timer".alarm_7_IN := FALSE;
   END_IF;
   //Формирование технологической защиты. Понижение разряжения в топке
   IF NOT "Protections_BLOCK".dP_in_furnance_min THEN
       "Protections".dP_in_furnance_min := "Alarm_Timer".alarm_7_Q;
   ELSE
       "Protections".dP_in_furnance_min := FALSE;
   END_IF;

   (*Понижение давления воздуха перед горелкой *)
   "Alarm_Timer".alarm_8_PT := T_CONV(INT_TO_DINT("Alarm_SP".TIME_P_air_before_burner_min) * 1000);
   IF "Alarm_Enable".P_air_before_burner_min THEN
       "Alarm_Timer".alarm_8_IN := "P_air_before_burner_min".Value OR ("P_air_burner".Value < "Alarm_SP".P_air_before_burner_min AND NOT "P_air_burner".Error_sensor AND "P_air_burner".N_module<>0);
       IF "Alarm_Timer".alarm_8_Q THEN
           "Alarm".P_air_before_burner_min := TRUE;
       END_IF;
   ELSE
       "Alarm_Timer".alarm_8_IN := FALSE;
   END_IF;
   //Формирование технологической защиты. Понижение давления воздуха перед горелкой
   IF NOT "Protections_BLOCK".P_air_before_burner_min THEN
       "Protections".P_air_before_burner_min := "Alarm_Timer".alarm_8_Q;
   ELSE
       "Protections".P_air_before_burner_min := FALSE;
   END_IF;

   (*Понижение уровня воды в барабане*)
   "Alarm_Timer".alarm_9_PT := T_CONV(INT_TO_DINT("Alarm_SP".TIME_L_water_min) * 1000);
   IF "Alarm_Enable".L_water_min THEN
       "Alarm_Timer".alarm_9_IN := "L_water_min".Value OR ("L_water".Value < "Alarm_SP".L_water_min AND NOT "L_water".Error_sensor AND "L_water".N_module <> 0);
       IF "Alarm_Timer".alarm_9_Q THEN
           "Alarm".L_water_min := TRUE;
       END_IF;
   ELSE
       "Alarm_Timer".alarm_9_IN := FALSE;
   END_IF;
   //Формирование технологической защиты. Понижение уровня воды в барабане
   IF NOT "Protections_BLOCK".L_water_min THEN
       "Protections".L_water_min := "Alarm_Timer".alarm_9_Q;
   ELSE
       "Protections".L_water_min := FALSE;
   END_IF;

   (*Повышение уровня воды в барабане*)
   "Alarm_Timer".alarm_10_PT := T_CONV(INT_TO_DINT("Alarm_SP".TIME_L_water_max) * 1000);
   IF "Alarm_Enable".L_water_max THEN
       "Alarm_Timer".alarm_10_IN := "L_water_max".Value OR ("L_water".Value > "Alarm_SP".L_water_max AND NOT "L_water".Error_sensor AND "L_water".N_module<>0);
       IF "Alarm_Timer".alarm_10_Q THEN
           "Alarm".L_water_max := TRUE;
       END_IF;
   ELSE
       "Alarm_Timer".alarm_10_IN := FALSE;
   END_IF;
   //Формирование технологической защиты. Повышение уровня воды в барабане
   IF NOT "Protections_BLOCK".L_water_max THEN
       "Protections".L_water_max := "Alarm_Timer".alarm_10_Q;
   ELSE
       "Protections".L_water_max := FALSE;
   END_IF;

   (*Повышение давления пара в барабане*)
   "Alarm_Timer".alarm_11_PT := T_CONV(INT_TO_DINT("Alarm_SP".TIME_P_steam_max) * 1000);
   IF "Alarm_Enable".P_steam_max THEN
       "Alarm_Timer".alarm_11_IN := "P_steam_max".Value OR ("P_steam".Value > "Alarm_SP".P_steam_max AND NOT "P_steam".Error_sensor AND "P_steam".N_module<>0);
       IF "Alarm_Timer".alarm_11_Q THEN
           "Alarm".P_steam_max := TRUE;
       END_IF;
   ELSE
       "Alarm_Timer".alarm_11_IN := FALSE;
   END_IF;
   //Формирование технологической защиты. Повышение давления пара в барабане
   IF NOT "Protections_BLOCK".P_steam_max THEN
       "Protections".P_steam_max := "Alarm_Timer".alarm_11_Q;
   ELSE
       "Protections".P_steam_max := FALSE;
   END_IF;

   (*Невоспламенение или погасание факела горелки котла*)
   "Alarm_Timer".alarm_12_PT := T_CONV(INT_TO_DINT("Alarm_SP".TIME_Not_flame_burner));
   IF "Alarm_Enable".Not_flame_burner THEN
       "Alarm_Timer".alarm_12_IN := NOT "Burner_flame".Value;
       IF "Alarm_Timer".alarm_12_Q THEN
           "Alarm".Not_flame_burner := TRUE;
       END_IF;
   ELSE
       "Alarm_Timer".alarm_12_IN := FALSE;
   END_IF;
   //Формирование технологической защиты. Невоспламенение или погасание факела горелки котла
   IF NOT "Protections_BLOCK".Not_flame_burner THEN
       "Protections".Not_flame_burner := "Alarm_Timer".alarm_12_Q;
   ELSE
       "Protections".Not_flame_burner := FALSE;
   END_IF;

   (*Нажата кнопка аварийного останова на панели оператора*)
   IF "Alarm_Enable".Alarm_stop_HMI THEN
       IF "FRONT".Btn_Alarm_stop_HMI THEN
           "Alarm".Alarm_stop_HMI := TRUE;
       END_IF;
   ELSE
       ;
   END_IF;
   //Формирование технологической защиты. Нажата кнопка аварийного останова на панели операторора
   IF NOT "Protections_BLOCK".Alarm_stop_HMI THEN
       "Protections".Alarm_stop_HMI := "FRONT".Btn_Alarm_stop_HMI;
   ELSE
       "Protections".Alarm_stop_HMI := FALSE;
   END_IF;

   (*Нажата кнопка аварийного останова на SCADA*)
   IF "Alarm_Enable".Alarm_stop_SCADA THEN
       IF "FRONT".Btn_Alarm_stop_SCADA THEN
           "Alarm".Alarm_stop_SCADA := TRUE;
       END_IF;
   ELSE
       ;
   END_IF;
   //Формирование технологической защиты. Нажата кнопка аварийного останова на SCADA
   IF NOT "Protections_BLOCK".Alarm_stop_SCADA THEN
       "Protections".Alarm_stop_SCADA := "FRONT".Btn_Alarm_stop_SCADA;
   ELSE
       "Protections".Alarm_stop_SCADA := FALSE;
   END_IF;

   (*СО2 порог 2*)
   "Alarm_Timer".alarm_13_PT := T_CONV(INT_TO_DINT("Alarm_SP".TIME_CO2));
   IF "Alarm_Enable".CO2 THEN
       "Alarm_Timer".alarm_13_IN := "CO_2".Value;
       IF "Alarm_Timer".alarm_13_Q THEN
           "Alarm".CO2 := TRUE;
       END_IF;
   ELSE
       "Alarm_Timer".alarm_13_IN := FALSE;
   END_IF;

   (*CH4*)
   "Alarm_Timer".alarm_14_PT := T_CONV(INT_TO_DINT("Alarm_SP".TIME_CH4));
   IF "Alarm_Enable".CH4 THEN
       "Alarm_Timer".alarm_14_IN := "CH4".Value;
       IF "Alarm_Timer".alarm_14_Q THEN
           "Alarm".CH4 := TRUE;
       END_IF;
   ELSE
       "Alarm_Timer".alarm_14_IN := FALSE;
   END_IF;

   (*ПРЕДУПРЕЖДЕНИЯ*)
   "TON_warning_1_DB".TON(IN := "Warning_Timer".warning_1_IN,
                          PT := "Warning_Timer".warning_1_PT,
                          Q => "Warning_Timer".warning_1_Q);
   "TON_warning_2_DB".TON(IN := "Warning_Timer".warning_2_IN,
                          PT := "Warning_Timer".warning_2_PT,
                          Q => "Warning_Timer".warning_2_Q);
   "TON_warning_3_DB".TON(IN := "Warning_Timer".warning_3_IN,
                          PT := "Warning_Timer".warning_3_PT,
                          Q => "Warning_Timer".warning_3_Q);
   "TON_warning_4_DB".TON(IN := "Warning_Timer".warning_4_IN,
                          PT := "Warning_Timer".warning_4_PT,
                          Q => "Warning_Timer".warning_4_Q);
   "TON_warning_5_DB".TON(IN := "Warning_Timer".warning_5_IN,
                          PT := "Warning_Timer".warning_5_PT,
                          Q => "Warning_Timer".warning_5_Q);
   "TON_warning_6_DB".TON(IN := "Warning_Timer".warning_6_IN,
                          PT := "Warning_Timer".warning_6_PT,
                          Q => "Warning_Timer".warning_6_Q);
   "TON_warning_7_DB".TON(IN := "Warning_Timer".warning_7_IN,
                          PT := "Warning_Timer".warning_7_PT,
                          Q => "Warning_Timer".warning_7_Q);
   "TON_warning_8_DB".TON(IN := "Warning_Timer".warning_8_IN,
                          PT := "Warning_Timer".warning_8_PT,
                          Q => "Warning_Timer".warning_8_Q);
   "TON_warning_9_DB".TON(IN := "Warning_Timer".warning_9_IN,
                          PT := "Warning_Timer".warning_9_PT,
                          Q => "Warning_Timer".warning_9_Q);
   "TON_warning_10".TON(IN := "Warning_Timer".warning_10_IN,
                        PT := "Warning_Timer".warning_10_PT,
                        Q => "Warning_Timer".warning_10_Q);

   (*Предупреждение. Неисправность датчика Температуры питательной воды перед экономайзером*)
   IF "T_water_before_economizer".N_module <> 0 AND "Warning_Enable".Sensor_T_water_before_economizer THEN
       "Warning".Sensor_T_water_before_economizer := "T_water_before_economizer".Error_sensor;
   ELSE
       "Warning".Sensor_T_water_before_economizer := FALSE;
   END_IF;

   (*Предупреждение. Неисправность датчика Температуры питательной воды после экономайзера*)
   IF "T_water_after_economizer".N_module <> 0 AND "Warning_Enable".Sensor_T_water_after_economizer THEN
       "Warning".Sensor_T_water_after_economizer := "T_water_after_economizer".Error_sensor;
   ELSE
       "Warning".Sensor_T_water_after_economizer := FALSE;
   END_IF;

   (*Предупреждение. Неисправность датчика перепада давления питательной воды на котел*)
   IF "dP_water_boiler".N_module <> 0 AND "Warning_Enable".Sensor_dP_water_boiler THEN
       "Warning".Sensor_dP_water_boiler := "dP_water_boiler".Error_sensor;
   ELSE
       "Warning".Sensor_dP_water_boiler := FALSE;
   END_IF;

   (*Предупреждение. Неисправность датчика Давления питательной воды до регулятора*)
   IF "P_water_before_regul".N_module <> 0 AND "Warning_Enable".Sensor_P_water_before_regul THEN
       "Warning".Sensor_P_water_before_regul := "P_water_before_regul".Error_sensor;
   ELSE
       "Warning".Sensor_P_water_before_regul := FALSE;
   END_IF;

   (*Предупреждение. Неисправность датчика Давления питательной воды после регулятора*)
   IF "P_water_after_regul".N_module <> 0 AND "Warning_Enable".Sensor_P_water_after_regul THEN
       "Warning".Sensor_P_water_after_regul := "P_water_after_regul".Error_sensor;
   ELSE
       "Warning".Sensor_P_water_after_regul := FALSE;
   END_IF;

   (*Предупреждение. Неисправность датчика Перепада давления пара в магистраль*)
   IF "dP_steam".N_module <> 0 AND "Warning_Enable".Sensor_dP_steam THEN
       "Warning".Sensor_dP_steam := "dP_steam".Error_sensor;
   ELSE
       "Warning".Sensor_dP_steam := FALSE;
   END_IF;

   (*Предупреждение. Неисправность датчика Давления пара в барабане*)
   IF "P_steam".N_module <> 0 AND "Warning_Enable".Sensor_P_steam THEN
       "Warning".Sensor_P_steam := "P_steam".Error_sensor;
   ELSE
       "Warning".Sensor_P_steam := FALSE;
   END_IF;

   (*Предупреждение. Неисправность датчика Разрежения в топке котла*)
   IF "dP_furnace_boiler".N_module <> 0 AND "Warning_Enable".Sensor_dP_furnace_boiler THEN
       "Warning".Sensor_dP_furnace_boiler := "dP_furnace_boiler".Error_sensor;
   ELSE
       "Warning".Sensor_dP_furnace_boiler := FALSE;
   END_IF;

   (*Предупреждение. Неисправность датчика Давления газа между ПЗК-1 и ПЗК-2*)
   IF "P_gas_between_PZK1_and_PZK2".N_module <> 0 AND "Warning_Enable".Sensor_P_gas_between_PZK1_and_PZK2 THEN
       "Warning".Sensor_P_gas_between_PZK1_and_PZK2 := "P_gas_between_PZK1_and_PZK2".Error_sensor;
   ELSE
       "Warning".Sensor_P_gas_between_PZK1_and_PZK2 := FALSE;
   END_IF;

